// TwinCAT 3 PLC project x_template_xPlc
// Title: x_template_xPlc
// Company: TcOpen.MTS
// ProjectVersion: 0.6.0.913
// ProgramVersion: 3.1.4023.0
// libraries:
//   Tc2_Standard, * (Beckhoff Automation GmbH)
//   Tc2_System, * (Beckhoff Automation GmbH)
//   Tc2_Utilities, * (Beckhoff Automation GmbH)
//   Tc3_Module, * (Beckhoff Automation GmbH)
//   TcoAbbRobotics, 0.12.0.111 (Vortex.Library)
//   TcoAbstractions, 0.12.0.111 (Vortex.Library)
//   TcoAimTtiPowerSupply, 0.12.0.111 (Vortex.Library)
//   TcoCognexVision, 0.12.0.111 (Vortex.Library)
//   TcoCore, 0.12.0.111 (Vortex.Library)
//   TcoData, 0.12.0.111 (Vortex.Library)
//   TcoDrivesBeckhoff, 0.12.0.111 (Vortex.Library)
//   TcoElements, 0.12.0.111 (Vortex.Library)
//   TcoInspectors, 0.12.0.111 (Vortex.Library)
//   TcoIo, 0.12.0.111 (Vortex.Library)
//   TcoKukaRobotics, 0.12.0.111 (Vortex.Library)
//   TcoMitsubishiRobotics, 0.12.0.111 (Vortex.Library)
//   TcoPneumatics, 0.12.0.111 (Vortex.Library)
//   TcoRexrothPress, 0.12.0.111 (Vortex.Library)
//   TcoTixonFeeding, 0.12.0.111 (Vortex.Library)
//   TcoUrRobotics, 0.12.0.111 (Vortex.Library)
//   TcoUtilities, 0.12.0.111 (Vortex.Library)
// project tree:
//   Abstractions/Components/ArrayRenderingExample/ SampleArrayToRender.TcDUT (not stored), SampleDataItem.TcDUT (not stored)
//   Abstractions/Components/MtsFeeding/Blisters/Plb/ TcoPlbPaletizator.TcPOU (not stored), TcoPlbPaletizator_Components.TcDUT (not stored), TcoPlbPaletizator_Config_v_1_x_x.TcDUT (not stored), TcoPlbPaletizator_Control_v_1_x_x.TcDUT (not stored), TcoPlbPaletizator_Positions.TcPOU (not stored), TcoPlbPaletizator_Status_v_1_x_x.TcDUT (not stored)
//   Abstractions/Components/MtsFeeding/Blisters/Plr/ TcoPlrPaletizator.TcPOU (not stored), TcoPlrPaletizator_Components.TcDUT (not stored), TcoPlrPaletizator_Config_v_1_x_x.TcDUT (not stored), TcoPlrPaletizator_Control_v_1_x_x.TcDUT (not stored), TcoPlrPaletizator_Status_v_1_x_x.TcDUT (not stored)
//   Abstractions/Components/MtsFeeding/Blisters/Pls/ TcoPlsPaletizator.TcPOU, TcoPlsPaletizator_Components.TcDUT, TcoPlsPaletizator_Config_v_1_x_x.TcDUT, TcoPlsPaletizator_Control_v_1_x_x.TcDUT (not stored), TcoPlsPaletizator_Status_v_1_x_x.TcDUT
//   Abstractions/Components/MtsFeeding/Blisters/ TcoFeeding_Config_v_1_x_x.TcDUT, TcoFeeding_Status_v_1_x_x.TcDUT
//   Abstractions/Components/MtsFeeding/OscilatingFeeder/ eTcoOscilatingConveyorOscilationModes.TcDUT (not stored), eTcoOscilatingConveyorStatus.TcDUT (not stored), TcoOscilatingConveyorFeeder.TcPOU (not stored), TcoOscilatingConveyorFeederComponents.TcDUT (not stored), TcoOscilatingConveyorFeeder_Config_v_1_x_x.TcDUT (not stored), TcoOscilatingConveyorFeeder_Control_v_1_x_x.TcDUT (not stored), TcoOscilatingConveyorFeeder_DesignerSpecificData.TcPOU (not stored), TcoOscilatingConveyorFeeder_PcToPlc.TcDUT (not stored), TcoOscilatingConveyorFeeder_PlcToPc.TcDUT (not stored), TcoOscilatingConveyorFeeder_Status_v_1_x_x.TcDUT (not stored)
//   Abstractions/Components/MtsFeeding/ TcoFeedingSequenceTask.TcPOU (not stored)
//   Abstractions/Components/Rework/ eReworkResults.TcDUT (not stored), ReworkData.TcDUT (not stored), ReworkInstructionTask.TcPOU (not stored)
//   Abstractions/Components/TS/EqTransfer/ eTcoEq2TransferConfiguration.TcDUT (not stored), eTcoEq2TransferHandlingMode.TcDUT (not stored), TcoEq2Transfer.TcPOU (not stored), TcoEq2TransferComponents.TcDUT (not stored), TcoEq2Transfer_Config.TcDUT (not stored), TcoEq2Transfer_Control.TcDUT (not stored), TcoEq2Transfer_Status.TcDUT (not stored)
//   Abstractions/Components/TS/RotaryTrabsferWithLift/ TcoLiftingRotaryTransfer.TcPOU (not stored), TcoLiftingRotaryTransferComponents.TcDUT (not stored), TcoLiftingRotaryTransfer_Config.TcDUT (not stored), TcoLiftingRotaryTransfer_Control.TcDUT (not stored), TcoLiftingRotaryTransfer_Status.TcDUT (not stored)
//   Abstractions/Components/TS/RotaryTransfer/ TcoRotaryTransfer.TcPOU (not stored), TcoRotaryTransferComponents.TcDUT (not stored), TcoRotaryTransfer_Config.TcDUT (not stored), TcoRotaryTransfer_Control.TcDUT (not stored), TcoRotaryTransfer_Status.TcDUT (not stored)
//   Abstractions/Components/TS/WorkPosition/ TcoTransferSystemComponent.TcPOU (not stored), TcoTransferSystemComponents.TcDUT (not stored), TcoTransferSystem_Config.TcDUT (not stored), TcoTransferSystem_Control.TcDUT (not stored), TcoTransferSystem_Status.TcDUT (not stored)
//   Abstractions/Components/WrappedComponent/ WrappedComponentExample.TcPOU (not stored), WrappedComponentExample_Config.TcDUT (not stored), WrappedComponentExample_Control.TcDUT (not stored), WrappedComponentExample_Status.TcDUT (not stored), WrappedComponentsExample.TcDUT (not stored)
//   Abstractions/CUBase/ CuBaseRecurringFail.TcDUT (not stored), CuBaseRecurringFailures.TcDUT (not stored), CUBase.TcPOU, CUBaseStatusInfo.TcDUT (not stored), CUBaseSettings.TcDUT (not stored), CUComponentsBase.TcDUT, ICUBase.TcIO (not stored), ICUTask.TcIO (not stored), OperatorInfo.TcDUT
//   Abstractions/CUBase/Data/ BasicCounterData.TcDUT (not stored), CuHeader.TcDUT (not stored), CUProcessDataBase.TcDUT (not stored), CUTechnologicalDataBase.TcDUT (not stored), eCUMode.TcDUT (not stored), eCUState.TcDUT (not stored), eDataEntityInvokeType.TcDUT (not stored), EntityHeader.TcDUT (not stored)
//   Abstractions/CUBase/RemoteTasks/ ProductionPlaner.TcPOU (not stored)
//   Abstractions/CUBase/Tasks/ CUBaseAutomat.TcPOU, CUBaseSuspend.TcPOU (not stored), CUBaseGround.TcPOU (not stored), CUBaseRecover.TcPOU (not stored)
//   Abstractions/Generic/LightTower/ TcoLightTower.TcPOU, TcoLightTower_Config.TcDUT (not stored), TcoLightTower_Info.TcDUT (not stored), TcoLightTower_Status.TcDUT (not stored)
//   Abstractions/Generic/NotificationPanel/ eIconType.TcDUT, Icon.TcDUT, NotificationPanel.TcPOU
//   Abstractions/Generic/TagsPairing/ eTagPairingAnswer.TcDUT (not stored), eTagPairingMode.TcDUT (not stored), eTagPairingStatus.TcDUT (not stored), PairTagTask.TcPOU (not stored), TagsPairing.TcDUT (not stored)
//   Abstractions/Safety/ControlButtons/ ITcoControlButtons.TcIO (not stored), TcoControlButtons.TcPOU (not stored), TcoControledZone_Info.TcDUT (not stored), VirtualButtons.TcDUT
//   Abstractions/Safety/ControlledZone/ TcoControlledZone.TcPOU, TcoControlledZoneActionTask.TcPOU (not stored), TcoControlledZone_Config.TcDUT (not stored), TcoControlledZone_Status.TcDUT (not stored)
//   Abstractions/Safety/ControlVoltage/ ITcoControlVoltage.TcIO (not stored), TcoControlVoltage.TcPOU (not stored)
//   Abstractions/Safety/DoorCircuit/ TcoDoorCircuit_Status.TcDUT (not stored), TcoDoorCircuit_Config.TcDUT (not stored), TcoDoorCircuit.TcPOU, ITcoDoorCircuit.TcIO (not stored)
//   Abstractions/Safety/Doors/ ITcoDoorLock.TcIO (not stored), TcoStandardDoor.TcPOU (not stored), TcoBasicDoor.TcPOU (not stored)
//   Abstractions/Safety/Estop/ TcoEmergencyStop.TcPOU (not stored)
//   Abstractions/Safety/KeyMode/ TcoKeyMode_Config.TcDUT (not stored), TcoKeyMode_Status.TcDUT (not stored), TcoKeyMode.TcPOU (not stored), ITcoKeyMode.TcIO (not stored)
//   Abstractions/Safety/KeyNormalService/ TcoKeyNormalService.TcPOU (not stored), ITcoKeyNormalSevice.TcIO (not stored)
//   Abstractions/TcoCore/ CycleTimeAnalitics.TcDUT (not stored), TcoCustomExportSeqData.TcDUT, TcoCustomStepDetails.TcDUT, TcoCustomTimeStruct.TcDUT, TcoInnerTask.TcPOU (not stored), TcoCustomSequencerObserver.TcPOU, TcoTaskedSequencer.TcPOU, TcoTaskedService.TcPOU (not stored)
//   Abstractions/Technology/ eStations.TcDUT
//   / MAIN.TcPOU (not stored), PlcTask.TcTTO (not stored)
//   Technology/CU00x/Automat/ CU00xAutomatParalell_1_Task.TcPOU, CU00xAutomatTask.TcPOU
//   Technology/CU00x/Components/ CU00xExamplesOfComponents.TcDUT (not stored), CU00xComponents.TcDUT
//   Technology/CU00x/Data/ CU00xTechnologicalData.TcDUT (not stored), CU00xDialogContent.TcPOU (not stored), CU00xProcessData.TcDUT
//   Technology/CU00x/Ground/ CU00xGroundTask.TcPOU (not stored)
//   Technology/CU00x/Manual/ CU00xManualTask.TcPOU (not stored)
//   Technology/CU00x/Positions/ CU00xTestMultiPositions.TcPOU (not stored), Cu00xTestPositions.TcPOU (not stored)
//   Technology/CU00x/Safety/Suspend/ CU00xSuspendTask.TcPOU
//   Technology/CU00x/Safety/Recover/ CU00xRecoverTask.TcPOU
//   Technology/Data/ InternalStorage.TcPOU, ProcessData.TcDUT, ProcessDataManager.TcPOU (not stored), TcoEntityBase.TcDUT (not stored), TechnologicalDataManager.TcPOU (not stored), TechnologyData.TcDUT
//   Technology/CU00x/ CU00x.TcPOU (not stored)
//   Technology/ Technology.TcPOU, TechnologyComponents.TcDUT
//   DUTs/IO/PDOs/ Device_State_F0482DC3.TcDUT (not stored), Device_Control_6258066A.TcDUT (not stored), Inputs_23559BB0.TcDUT (not stored), Outputs_FC2FACAD.TcDUT (not stored), Modules_85784B27.TcDUT (not stored), Channel_830843C1.TcDUT (not stored), Channel_42CA91F7.TcDUT (not stored)
//   DUTs/IO/Boxes/ EK1200_013D0B49.TcDUT (not stored), EK1122_1FC0878B.TcDUT (not stored), AES_510494FB.TcDUT (not stored), EPP1322_1FC0878B.TcDUT (not stored), EPP1809_32157CFD.TcDUT (not stored), EPP1008_78E8D3DD.TcDUT (not stored), EL1809_32157CFD.TcDUT (not stored), EL2809_2B6483BD.TcDUT (not stored), EL9011_D65D3D32.TcDUT (not stored)
//   DUTs/IO/Devices/ SyncUnitTasks_4BE01469.TcDUT (not stored), SyncUnits_67D36DDA.TcDUT (not stored)
//   DUTs/IO/Topology/ EK_E812B8FA.TcDUT (not stored), EC_4E5C738F.TcDUT (not stored), EC_245FBB9A.TcDUT (not stored)
//   GVLs/ GVL_iXlinker.TcGVL (not stored)
// real-time tasks:
//   TASK PlcTask: cycle T#10ms, priority 20, ADS port 350
//   TASK PlcTask1: cycle T#10ms, priority 21, ADS port 351
// I/O:
//   DEVICE EC1 (disabled), AmsNetId 192.168.4.1.7.1
//     (EK1200) [EK1200-5000 EtherCAT Power supply (2A E-Bus)]
//       EC (EK1122) [EK1122 2 port EtherCAT junction]
//       PN (EL6631) [EL6631 PROFINET IO Controller]
//       IA1 (EL1809) [EL1809 16Ch. Dig. Input 24V, 3ms]
//       QA1 (EL2809) [EL2809 16Ch. Dig. Output 24V, 0.5A]
//       Term 6 (EL4004) [EL4004 4Ch. Ana. Output 0-10V, 12bit]
//       Term 7 (EL7342) [EL7342 2Ch. DC motor output stage (50V, 3.5A)]
//       Term 8 (EL4004) [EL4004 4Ch. Ana. Output 0-10V, 12bit]
//       Term 9 (EL6001) [EL6001 Interface (RS232)]
//       Term 13 (EL9011) [EL9011 End Terminal]
//   DEVICE EC (disabled), AmsNetId 192.168.4.1.2.1
//     EC [EK1200-5000 EtherCAT Power supply (2A E-Bus)]
//       EK [EK1122 2 port EtherCAT junction]
//         PNEU [AES Fieldbus Coupler Gen2]
//           modules: Modules
//         AB [EPP1322-0001 3 port EtherCAT P gateway]
//         AB21 [EPP1809-0021 16 Ch. Dig. Input 24V, 3ms, M8]
//         AB22 [EPP1809-0021 16 Ch. Dig. Input 24V, 3ms, M8]
//         AB23 [EPP1008-0001 8 Ch. Dig. Input 24V, 3ms, M8]
//         AB24 [EPP1008-0001 8 Ch. Dig. Input 24V, 3ms, M8]
//       IA1 [EL1809 16Ch. Dig. Input 24V, 3ms]
//       QA1 [EL2809-0015 16Ch. Dig. Output 24V DC, 0.35A, not short-circuit proof]
//       Term 11 (EL9011) [EL9011 End Terminal]
// variable links:
//   x_template_xPlc/x_template_xPlc Instance <-> EC
//     PlcTask Inputs/GVL_iXlinker.EC.InfoData.AmsNetId <-> InfoData/AmsNetId
//     PlcTask Inputs/GVL_iXlinker.EC.InfoData.CfgSlaveCount <-> InfoData/CfgSlaveCount
//     PlcTask Inputs/GVL_iXlinker.EC.InfoData.ChangeCount <-> InfoData/ChangeCount
//     PlcTask Inputs/GVL_iXlinker.EC.InfoData.DevId <-> InfoData/DevId
//     PlcTask Inputs/GVL_iXlinker.EC.Inputs.DevState <-> Inputs/DevState
//     PlcTask Inputs/GVL_iXlinker.EC.Inputs.Frm0InputToggle <-> Inputs/Frm0InputToggle
//     PlcTask Inputs/GVL_iXlinker.EC.Inputs.Frm0State <-> Inputs/Frm0State
//     PlcTask Inputs/GVL_iXlinker.EC.Inputs.Frm0WcState <-> Inputs/Frm0WcState
//     PlcTask Inputs/GVL_iXlinker.EC.Inputs.SlaveCount <-> Inputs/SlaveCount
//     PlcTask Outputs/GVL_iXlinker.EC.Outputs.DevCtrl <-> Outputs/DevCtrl
//     PlcTask Outputs/GVL_iXlinker.EC.Outputs.Frm0Ctrl <-> Outputs/Frm0Ctrl
//     PlcTask Outputs/GVL_iXlinker.EC.Outputs.Frm0WcCtrl <-> Outputs/Frm0WcCtrl
//   x_template_xPlc/x_template_xPlc Instance <-> EC/EC/EK
//     PlcTask Inputs/GVL_iXlinker.EC.EC.EK.InfoData.State <-> InfoData/State
//   x_template_xPlc/x_template_xPlc Instance <-> EC/EC/EK/AB
//     PlcTask Inputs/GVL_iXlinker.EC.EC.EK.AB.InfoData.State <-> InfoData/State
//   x_template_xPlc/x_template_xPlc Instance <-> EC/EC/EK/AB21
//     PlcTask Inputs/GVL_iXlinker.EC.EC.EK.AB21.Channel_{1..16}.Input <-> Channel {1..16}/Input  (16 links)
//     PlcTask Inputs/GVL_iXlinker.EC.EC.EK.AB21.InfoData.State <-> InfoData/State
//     PlcTask Inputs/GVL_iXlinker.EC.EC.EK.AB21.WcState.InputToggle <-> WcState/InputToggle
//     PlcTask Inputs/GVL_iXlinker.EC.EC.EK.AB21.WcState.WcState <-> WcState/WcState
//   x_template_xPlc/x_template_xPlc Instance <-> EC/EC/EK/AB22
//     PlcTask Inputs/GVL_iXlinker.EC.EC.EK.AB22.Channel_{1..16}.Input <-> Channel {1..16}/Input  (16 links)
//     PlcTask Inputs/GVL_iXlinker.EC.EC.EK.AB22.InfoData.State <-> InfoData/State
//     PlcTask Inputs/GVL_iXlinker.EC.EC.EK.AB22.WcState.InputToggle <-> WcState/InputToggle
//     PlcTask Inputs/GVL_iXlinker.EC.EC.EK.AB22.WcState.WcState <-> WcState/WcState
//   x_template_xPlc/x_template_xPlc Instance <-> EC/EC/EK/AB23
//     PlcTask Inputs/GVL_iXlinker.EC.EC.EK.AB23.Channel_{1..8}.Input <-> Channel {1..8}/Input  (8 links)
//     PlcTask Inputs/GVL_iXlinker.EC.EC.EK.AB23.InfoData.State <-> InfoData/State
//     PlcTask Inputs/GVL_iXlinker.EC.EC.EK.AB23.WcState.InputToggle <-> WcState/InputToggle
//     PlcTask Inputs/GVL_iXlinker.EC.EC.EK.AB23.WcState.WcState <-> WcState/WcState
//   x_template_xPlc/x_template_xPlc Instance <-> EC/EC/EK/AB24
//     PlcTask Inputs/GVL_iXlinker.EC.EC.EK.AB24.Channel_{1..8}.Input <-> Channel {1..8}/Input  (8 links)
//     PlcTask Inputs/GVL_iXlinker.EC.EC.EK.AB24.InfoData.State <-> InfoData/State
//     PlcTask Inputs/GVL_iXlinker.EC.EC.EK.AB24.WcState.InputToggle <-> WcState/InputToggle
//     PlcTask Inputs/GVL_iXlinker.EC.EC.EK.AB24.WcState.WcState <-> WcState/WcState
//   x_template_xPlc/x_template_xPlc Instance <-> EC/EC/EK/PNEU
//     PlcTask Inputs/GVL_iXlinker.EC.EC.EK.PNEU.Device_State.CommonValve <-> Device_State/CommonValve
//     PlcTask Inputs/GVL_iXlinker.EC.EC.EK.PNEU.Device_State.Configuration_Error_IO_Module <-> Device_State/Configuration Error IO-Module
//     PlcTask Inputs/GVL_iXlinker.EC.EC.EK.PNEU.Device_State.Configuration_Error_Valve <-> Device_State/Configuration Error Valve
//     PlcTask Inputs/GVL_iXlinker.EC.EC.EK.PNEU.Device_State.Configuratipn_Error_SLS <-> Device_State/Configuratipn Error SLS
//     PlcTask Inputs/GVL_iXlinker.EC.EC.EK.PNEU.Device_State.Count_IO_Module_to_big <-> Device_State/Count IO-Module to big
//     PlcTask Inputs/GVL_iXlinker.EC.EC.EK.PNEU.Device_State.Heardbeat_x <-> Device_State/Heardbeat
//     PlcTask Inputs/GVL_iXlinker.EC.EC.EK.PNEU.Device_State.IO_1_8 <-> Device_State/IO:1-8
//     PlcTask Inputs/GVL_iXlinker.EC.EC.EK.PNEU.Device_State.IO_9_10 <-> Device_State/IO:9-10
//     PlcTask Inputs/GVL_iXlinker.EC.EC.EK.PNEU.Device_State.Switchcounter_Error <-> Device_State/Switchcounter Error
//     PlcTask Inputs/GVL_iXlinker.EC.EC.EK.PNEU.Device_State.UA_OFF <-> Device_State/UA OFF
//     PlcTask Inputs/GVL_iXlinker.EC.EC.EK.PNEU.Device_State.UL_OFF <-> Device_State/UL OFF
//     PlcTask Inputs/GVL_iXlinker.EC.EC.EK.PNEU.Device_State.Undervoltage_5V <-> Device_State/Undervoltage 5V
//     PlcTask Inputs/GVL_iXlinker.EC.EC.EK.PNEU.Device_State.Undervoltage_UA <-> Device_State/Undervoltage UA
//     PlcTask Inputs/GVL_iXlinker.EC.EC.EK.PNEU.Device_State.Undervoltage_UL <-> Device_State/Undervoltage UL
//     PlcTask Inputs/GVL_iXlinker.EC.EC.EK.PNEU.Device_State.Unknown_Module_ID <-> Device_State/Unknown Module ID
//     PlcTask Inputs/GVL_iXlinker.EC.EC.EK.PNEU.Device_State.ValveExtSupplyDiag_1_6 <-> Device_State/ValveExtSupplyDiag:1-6
//     PlcTask Inputs/GVL_iXlinker.EC.EC.EK.PNEU.InfoData.AdsAddr <-> InfoData/AdsAddr
//     PlcTask Inputs/GVL_iXlinker.EC.EC.EK.PNEU.InfoData.State <-> InfoData/State
//     PlcTask Inputs/GVL_iXlinker.EC.EC.EK.PNEU.Modules.Inputs.digital_Data_I[{0..31}] <-> Modules/Inputs/digital Data I_{0..31}  (32 links)
//     PlcTask Inputs/GVL_iXlinker.EC.EC.EK.PNEU.WcState.InputToggle <-> WcState/InputToggle
//     PlcTask Inputs/GVL_iXlinker.EC.EC.EK.PNEU.WcState.WcState <-> WcState/WcState
//     PlcTask Outputs/GVL_iXlinker.EC.EC.EK.PNEU.Device_Control.Default_Modul_Control <-> Device_Control/Default_Modul_Control
//     PlcTask Outputs/GVL_iXlinker.EC.EC.EK.PNEU.Device_Control.Freeze_Output <-> Device_Control/Freeze Output
//     PlcTask Outputs/GVL_iXlinker.EC.EC.EK.PNEU.Device_Control.HL_Swap <-> Device_Control/HL_Swap
//     PlcTask Outputs/GVL_iXlinker.EC.EC.EK.PNEU.Device_Control.Web_App_Disable <-> Device_Control/Web App Disable
//     PlcTask Outputs/GVL_iXlinker.EC.EC.EK.PNEU.Modules.Outputs.digital_Data_O[{0..31}] <-> Modules/Outputs/digital Data O_{0..31}  (32 links)
//   x_template_xPlc/x_template_xPlc Instance <-> EC/EC/IA1
//     PlcTask Inputs/GVL_iXlinker.EC.EC.IA1.Channel_{1..16}.Input <-> Channel {1..16}/Input  (16 links)
//     PlcTask Inputs/GVL_iXlinker.EC.EC.IA1.InfoData.State <-> InfoData/State
//     PlcTask Inputs/GVL_iXlinker.EC.EC.IA1.WcState.InputToggle <-> WcState/InputToggle
//     PlcTask Inputs/GVL_iXlinker.EC.EC.IA1.WcState.WcState <-> WcState/WcState
//   x_template_xPlc/x_template_xPlc Instance <-> EC/EC/QA1
//     PlcTask Inputs/GVL_iXlinker.EC.EC.QA1.InfoData.State <-> InfoData/State
//     PlcTask Inputs/GVL_iXlinker.EC.EC.QA1.WcState.WcState <-> WcState/WcState
//     PlcTask Outputs/GVL_iXlinker.EC.EC.QA1.Channel_{1..16}.Output <-> Channel {1..16}/Output  (16 links)

// ---- Abstractions/Components/MtsFeeding/Blisters/Pls/TcoPlsPaletizator_Components.TcDUT
TYPE TcoPlsPaletizator_Components EXTENDS TcoCore.TcoStruct:
STRUCT
	
	{attribute wpf [Container(Layout.Stack)]}
	{attribute addProperty Name "(I1) <#Blister present in entry slide#>"}
	I1_PresentBlisterEntry : TcoElements.TcoDi(THISSTRUCT);
	
	{attribute addProperty Name "(I2) <#Gap detected between blisters#>"}
	I2_PresentBlisterEntryEmptySpace : TcoElements.TcoDi(THISSTRUCT);
	
	{attribute addProperty Name "(I3) <#Blister feeder empty#>"}
	I3_PresentBlistersInBufferEmpty : TcoElements.TcoDi(THISSTRUCT);

	
	{attribute addProperty Name "(I4) <#Blister in working position#>"}
	I4_PresentBlisterInWorkingPos : TcoElements.TcoDi(THISSTRUCT);
		
	{attribute addProperty Name "(I5) <#Output blister not on slide conveyor#>"}
	I5_OutBlistersIsThrowedCorrectly : TcoElements.TcoDi(THISSTRUCT);
	
	{attribute addProperty Name "(I6) <#Output blister present in elevator#>"}
	I6_OutBlistersLisftSignal : TcoElements.TcoDi(THISSTRUCT);
	
	{attribute addProperty Name "(I7) <#Output blister above buffer#>"}
	I7_OutBlistersIsAboveOutBuffer : TcoElements.TcoDi(THISSTRUCT);
	
	{attribute addProperty Name "(I8) <#Output container full#>"}
	I8_OutBlistersBufferIsFull : TcoElements.TcoDi(THISSTRUCT);
	
	
	{attribute wpf [Container(Layout.Stack)]}
	{attribute addProperty Name "(P1) <#Entry blister lift#>"}
	P1_VerticalSepareEntryBlisters : TcoPneumatics.TcoCylinder(THISSTRUCT);
	
	{attribute addProperty Name "(P2) <#Entry blister lift#>"}
	P2_VerticalSepareEntryBlisters : TcoPneumatics.TcoCylinder(THISSTRUCT);
	
	{attribute addProperty Name "(P3) (P3.1) <#Entry blister slide#>"}
	P3_HorizontalSepareEntryBlisters : TcoPneumatics.TcoDoubleCylinder(THISSTRUCT);
		
	{attribute addProperty Name "(P4) <#Entry blister feed#>"}
	P4_FeedEntryBlister :TcoPneumatics.TcoCylinder(THISSTRUCT);
	
	{attribute addProperty Name "(P5) (P5.1) <#Output blister slide#>"}
	P5_HorizontalSepareOutBlisters : TcoPneumatics.TcoDoubleCylinder(THISSTRUCT);
	
	{attribute addProperty Name "(P6) <#Output blister lift#>"}
	P6_VerticalSepareOutBlister : TcoPneumatics.TcoCylinder(THISSTRUCT);
	
	{attribute addProperty Name "(P7) <#Entry blister support#>"}
	P7_SupportEntryBlister : TcoPneumatics.TcoCylinder(THISSTRUCT);
	
	{attribute addProperty Name "(P8) (P8.1) <#Entry blister side clamp#>"}
	P8_FixEntryBlisterSide : TcoPneumatics.TcoDoubleCylinder(THISSTRUCT);
	
	{attribute addProperty Name "(P9) (P9.1) <#Entry blister top clamp#>"}
	P9_LockEntryBlisterTop : TcoPneumatics.TcoDoubleCylinder(THISSTRUCT);
	
	{attribute addProperty Name "(P10) (P10.1) <#Entry blister separator#>"}
	P10_HoldEntrySepareOutBlister : TcoPneumatics.TcoDoubleCylinder(THISSTRUCT);
	
	
	
	{attribute wpf [Container(Layout.Stack,"Vseobecne")]}
	
	{attribute addProperty Name "(Q1) <#Warning signalisation#> R"}
	Q1_AttentionSignalisationR : TcoElements.TcoDo(THISSTRUCT);
	{attribute addProperty Name "(Q2) <#Warning signalisation#> G"}
	Q2_AttentionSignalisationG : TcoElements.TcoDo(THISSTRUCT);
	{attribute addProperty Name "(Q3) <#Warning signalisation#> B"}
	Q3_AttentionSignalisationB : TcoElements.TcoDo(THISSTRUCT);

	
	
END_STRUCT
END_TYPE

// ---- Abstractions/Components/MtsFeeding/Blisters/Pls/TcoPlsPaletizator_Config_v_1_x_x.TcDUT
TYPE
    TcoPlsPaletizator_Config_v_1_x_x EXTENDS TcoFeeding_Config_v_1_x_x :
    STRUCT

		
		
        {attribute addProperty Name "<#Locking of the blister from above inactive (P9)(P9.1) is not present#>"}
		LockBlisterInPickPosInactive : BOOL;
		
		{attribute addProperty Name "<#Separation of entry blisters inactive (P10)(P10.1) is not present#>"}
		SepareBlistersAtEntryInactive : BOOL;

    END_STRUCT
END_TYPE

// ---- Abstractions/Components/MtsFeeding/Blisters/Pls/TcoPlsPaletizator_Status_v_1_x_x.TcDUT
TYPE
    TcoPlsPaletizator_Status_v_1_x_x EXTENDS TcoFeeding_Status_v_1_x_x:
    STRUCT

        {attribute addProperty Name "<#Refill required#>"}
		EntryBufferEmpty:BOOL;
		
		{attribute addProperty Name "<#Blister ready#>"}
        BlisterReady : BOOL;
		
		{attribute addProperty Name "<#Empty blisters removal required#>"}
        OutBufferFull : BOOL;
    END_STRUCT
END_TYPE

// ---- Abstractions/Components/MtsFeeding/Blisters/TcoFeeding_Config_v_1_x_x.TcDUT
TYPE
    TcoFeeding_Config_v_1_x_x EXTENDS TcoCore.TcoStruct :
    STRUCT

		{attribute addProperty Name "<#Info delay#>"}
        InfoTime : TIME := T#5S;
		{attribute addProperty Name "<#Error delay#>"}
        ErrorTime : TIME := T#0S;
        {attribute addProperty Name "<#Stabilisation time#>"}
        StabilisationTime : TIME := T#500MS;
        {attribute addProperty Name "<#Blink period#> "}
        BlinkTime : TIME := T#500MS;

        {attribute addProperty Name "<#Safety disable duration#> "}
        TimeToDisableSafety : TIME := T#10S;

        {attribute addProperty Name "<#Step mode managable from outside#> (SetSequencesToStep)"}
        StepModeManagableFromOutside : BOOL;

    END_STRUCT
END_TYPE

// ---- Abstractions/Components/MtsFeeding/Blisters/TcoFeeding_Status_v_1_x_x.TcDUT
TYPE
    TcoFeeding_Status_v_1_x_x EXTENDS TcoCore.TcoStruct :
    STRUCT

	
		{attribute addProperty Name "<#Action#>"}
        ActionDescription : STRING;
		
		{attribute addProperty Name "<#Safety conditon met#>"}
        SafeCondition : BOOL;

    END_STRUCT
END_TYPE

// ---- Abstractions/CUBase/CUComponentsBase.TcDUT
TYPE
    CUComponentsBase EXTENDS TcoCore.TcoStruct :
    STRUCT
       	{attribute wpf [Container(Layout.Stack)]}
		{attribute clr [RenderIgnore()]}
        DummyCylinder : TcoPneumatics.TcoCylinder(THISSTRUCT);
		{attribute clr [RenderIgnore()]}
        DummyDi : TcoElements.TcoDi(THISSTRUCT);
		{attribute clr [RenderIgnore()]}
        DummyDo : TcoElements.TcoDo(THISSTRUCT);
    END_STRUCT
END_TYPE

// ---- Abstractions/CUBase/OperatorInfo.TcDUT
TYPE OperatorInfo EXTENDS TcoCore.TcoStruct :
STRUCT
	UserName : STRING(255);
	
END_STRUCT
END_TYPE

// ---- Abstractions/Generic/NotificationPanel/eIconType.TcDUT
{attribute 'qualified_only'}
{attribute 'strict'}
{attribute 'to_string'}
TYPE 
	eIconType : 
(
	None                 := 0,
	ControlVoltage       := 10,
	AirPressure          := 20,
	EmergencyStop        := 30,
	SafetyDoor           := 40,
	DoorClosed           := 50,
	DoorLocked           := 60,
	AutomatAllowed       := 70,
	ProcessDataLoaded    := 80,
	TechnologyDataLoaded := 90,
	OpticBarrier         := 100,
	Robot                := 110,
	PlcConnection        := 120
);
END_TYPE

// ---- Abstractions/Generic/NotificationPanel/Icon.TcDUT
TYPE Icon :
STRUCT
	Title : STRING;
	IconType : STRING;
	Signal : BOOL;
	BlinkingEnabled : BOOL := FALSE;
	EnableRedIcon : BOOL := TRUE;
	
	///used internally
	SignalBlink : BOOL;
END_STRUCT
END_TYPE

// ---- Abstractions/Safety/ControlButtons/VirtualButtons.TcDUT
TYPE VirtualButtons :
STRUCT
	StartButton:BOOL;
	StopButton:BOOL;
	GroundButton:BOOL;
	AutomatButton:BOOL;

	StartLight : BOOL;
	StopLight : BOOL;
END_STRUCT
END_TYPE

// ---- Abstractions/TcoCore/TcoCustomExportSeqData.TcDUT
TYPE
    TcoCustomExportSeqData :
    STRUCT

        Steps : ARRAY[0..TcoCustomSequencerObserver.MAX_STEPS] OF TcoCustomStepDetails;
        CycleId : STRING(254);
        CuId : UINT;
        StartTime : TcoCustomTimeStruct;
        EndTime : TcoCustomTimeStruct;
    END_STRUCT
END_TYPE

// ---- Abstractions/TcoCore/TcoCustomStepDetails.TcDUT

TYPE TcoCustomStepDetails :
STRUCT

	{attribute addProperty Name "<#Step ID#>"}
	ID: INT;

	{attribute addProperty Name "<#Step description#>"}
	Description: STRING(254);

	{attribute addProperty Name "<#Step duration#>"}
	Duration : TIME;
	
	{attribute addProperty Name "<#Time Stamp Struct#>"}
	TimeStamp : TcoCustomTimeStruct;
	
END_STRUCT
END_TYPE

// ---- Abstractions/TcoCore/TcoCustomTimeStruct.TcDUT
TYPE
    TcoCustomTimeStruct :
    STRUCT
        Year : WORD;
        Month : WORD;

        Day : WORD;
        Hour : WORD;
        Minute : WORD;
        Second : WORD;
        Milliseconds : WORD;
    END_STRUCT
END_TYPE

// ---- Abstractions/Technology/eStations.TcDUT
{attribute 'qualified_only'}
{attribute 'strict'}
TYPE
    eStations :
    (
		CU00x := 100,
       CU010  := 1,
        CU020  := 2,
        CU030  := 3,
        CU040  := 4,
        CU050  := 5,
        ST_6  := 6,
        ST_7  := 7,
        ST_8  := 8,
        ST_9  := 9,
        ST_10 := 10,
        ST_11 := 11,
        ST_12 := 12,
        ST_13 := 13,
        ST_14 := 14,
        ST_15 := 15,
        ST_16 := 16,
        ST_17 := 17,
        ST_18 := 18,
        ST_19 := 19,
        ST_20 := 20,
        NONE  := 32767
    );
END_TYPE

// ---- Technology/Data/ProcessData.TcDUT
{attribute clr [Container(Layout.Tabs)]}
TYPE
    ProcessData EXTENDS TcoEntityBase :
    STRUCT

        {attribute addProperty Name "<#Entity header#>"}
        EntityHeader : EntityHeader     := (Parent := THISSTRUCT);
		{attribute addProperty Name "<#CU00x#>"}
		{attribute clr [Container(Layout.Stack)]}
        CU00x : CU00xProcessData := (Parent := THISSTRUCT);
		
//		
		CU010 : CU010ProcessData := (Parent := THISSTRUCT);
		CU020 : CU020ProcessData := (Parent := THISSTRUCT);
		CU030 : CU030ProcessData := (Parent := THISSTRUCT);
		CU040 : CU040ProcessData := (Parent := THISSTRUCT);
		CU050 : CU050ProcessData := (Parent := THISSTRUCT);
    END_STRUCT
END_TYPE

// ---- Technology/CU00x/Components/CU00xComponents.TcDUT
{attribute wpf [Container(Layout.Tabs)]}
TYPE
    CU00xComponents EXTENDS CUComponentsBase :
    STRUCT
		{attribute wpf [Container(Layout.Stack)]}
		{attribute wpf [Group(Layout.Scroll)]}
		{attribute addProperty Name "Supplu TTI QL"}
     	Supply : TcoAimTtiPowerSupply.TcoQl355P_v_1_x_x (THISSTRUCT);
		{attribute wpf [Container(Layout.Stack)]}
		PairTagTask: PairTagTask(THISSTRUCT);
		{attribute wpf [Container(Layout.Stack)]}
		{attribute addProperty Name "<#ReworkInstruction#>"}
		ReworkInstructionTask : ReworkInstructionTask(THISSTRUCT);
		{attribute wpf [Container(Layout.Stack,"DRIVES AND MANIPULATORS")]}	
		{attribute wpf [Group(Layout.Scroll)]}
		{attribute addProperty Name "MultiAxis"}
     	MultiAxis : TcoDrivesBeckhoff.TcoMultiAxis(THISSTRUCT);
		{attribute addProperty Name "Single Axis"}
     	SingleAxis : TcoDrivesBeckhoff.TcoSingleAxis(THISSTRUCT);
		{attribute addProperty Name "Simple drive"}
     	SimpleDrive : TcoDrivesBeckhoff.TcoDriveSimple(THISSTRUCT);
		
		{attribute wpf [Container(Layout.Stack,"VISION")]}	
		{attribute wpf [Group(Layout.Scroll)]}
		{attribute addProperty Name "Dataman"}
     	Dmc : TcoCognexVision.TcoDataman_v_5_x_x(THISSTRUCT);
		{attribute addProperty Name "Insight"}
     	Cam : TcoCognexVision.TcoInsight_v_5_x_x(THISSTRUCT);

	
		{attribute wpf [Container(Layout.Stack,"ROBOTICS")]}	
		{attribute wpf [Group(Layout.Scroll)]}
		{attribute addProperty Name "Abb IRC 5"}
     	AbbIrc5 : TcoAbbRobotics.TcoIrc5_v_1_x_x(THISSTRUCT);
		{attribute addProperty Name "Abb Omnicore"}
     	AbbOmnicore : TcoAbbRobotics.TcoOmnicore_v_1_x_x(THISSTRUCT);
		
		{attribute addProperty Name "Mitshubishi Cr series"}
     	MitshubishiCr: TcoMitsubishiRobotics.TcoCr800_v_1_x_x(THISSTRUCT);
		{attribute addProperty Name "UR CB series"}
     	UrCb3:  TcoUrRobotics.TcoUrCb3_v_3_x_x(THISSTRUCT);
		{attribute addProperty Name "Ur E series"}
     	UrEseries: TcoUrRobotics.TcoUrEseries_v_5_x_x(THISSTRUCT);
		
		{attribute addProperty Name "Kuka Krc4"}
     	KukaKrc4: TcoKukaRobotics.TcoKrc4_v_5_x_x(THISSTRUCT);
		
		{attribute wpf [Container(Layout.Stack,"TIXONS")]}	
		{attribute wpf [Group(Layout.Scroll)]}
		{attribute addProperty Name "Tixon Vibro"}
     	TixonVibro : TcoTixonFeeding.TcoTixonVibro_v_1_x_x(THISSTRUCT);
		{attribute addProperty Name "Tixon Step"}
     	TixonStep : TcoTixonFeeding.TcoTixonStep_v_1_x_x(THISSTRUCT);
		
		{attribute addProperty Name "Tixon Pick Vibro"}
     	TixonPickVibro : TcoTixonFeeding.TcoTixonPickVibro_v_1_x_x(THISSTRUCT);
		{attribute addProperty Name "Tixon Pick Step"}
     	TixonPickStep : TcoTixonFeeding.TcoTixonPickStep_v_1_x_x(THISSTRUCT);
			
		{attribute wpf [Container(Layout.Stack,"MtsFeeding")]}	
		{attribute wpf [Group(Layout.Scroll)]}
		PlsPaletizator:TcoPlsPaletizator(THISSTRUCT);	
		{attribute clr [RenderIgnore()]}
		PlsPaletizatorComponents:TcoPlsPaletizator_Components := (Parent := THISSTRUCT);  
		
		{attribute wpf [Group(Layout.Scroll)]}
		PlrPaletizator:TcoPlrPaletizator(THISSTRUCT);	
		{attribute clr [RenderIgnore()]}
		PlrPaletizatorComponents:TcoPlrPaletizator_Components := (Parent := THISSTRUCT);  
		
		{attribute wpf [Group(Layout.Scroll)]}
		PlbPaletizator:TcoPlbPaletizator(THISSTRUCT);	
		{attribute clr [RenderIgnore()]}
		PlbPaletizatorComponents:TcoPlbPaletizator_Components := (Parent := THISSTRUCT);  
		
		
		{attribute wpf [Container(Layout.Stack)]}
        {attribute wpf [Group(Layout.Scroll)]}
        OscilatingFeeder : TcoOscilatingConveyorFeeder(THISSTRUCT);
        {attribute clr [RenderIgnore()]}
        OscilatingFeederComponents : TcoOscilatingConveyorFeederComponents := (Parent := THISSTRUCT);

		
		{attribute wpf [Container(Layout.Stack,"Wrapped component example")]}	
		{attribute wpf [Group(Layout.Scroll)]}
		PickAndPlace:WrappedComponentExample(THISSTRUCT);
		{attribute wpf [Container(Layout.Stack,"Wrapped component struct")]}	
		PickAndPlaceCompoennts:WrappedComponentsExample := (Parent := THISSTRUCT);  

		{attribute addProperty Name "GROUP 1"}
		Group1 : CU00xExamplesOfComponents := (Parent := THISSTRUCT);  
		{attribute addProperty Name "GROUP 2"}
		Group2 : CU00xExamplesOfComponents := (Parent := THISSTRUCT); 
 
		
		
		{attribute wpf [Container(Layout.Stack,"PanaTrace")]}	
		{attribute wpf [Group(Layout.Scroll)]}
		PanaTrace:TcoPscPanaTrace(THISSTRUCT);
    END_STRUCT
END_TYPE

// ---- Technology/CU00x/Data/CU00xProcessData.TcDUT
TYPE
    CU00xProcessData EXTENDS CUProcessDataBase :
    STRUCT
		{attribute wpf [Container(Layout.Stack)]}
		{attribute addProperty Name "Bolt present inspection"}
        BoltPresenceInspector : TcoInspectors.TcoDigitalInspector(THISSTRUCT);
		{attribute addProperty Name "Bolt Dimension inspection"}
		BoltDimensionPresenceInspector : TcoInspectors.TcoAnalogueInspector(THISSTRUCT);
		{attribute addProperty Name "Bolt code inspection"}
		BoltDatacodePresenceInspector : TcoInspectors.TcoDataInspector(THISSTRUCT);
		

		{attribute addProperty Name "Dimension inspection 1"}
        Dim_Inspector_1 : TcoInspectors.TcoAnalogueInspector(THISSTRUCT);
		{attribute addProperty Name "Dimension inspection 2"}
        Dim_Inspector_2 : TcoInspectors.TcoAnalogueInspector(THISSTRUCT);
		{attribute addProperty Name "Dimension inspection 3"}
		Dim_Inspector_3 : TcoInspectors.TcoAnalogueInspector(THISSTRUCT);
		{attribute addProperty Name "Dimension inspection 4"}
        Dim_Inspector_4 : TcoInspectors.TcoAnalogueInspector(THISSTRUCT);
		{attribute addProperty Name "Dimension inspection 5"}
        Dim_Inspector_5 : TcoInspectors.TcoAnalogueInspector(THISSTRUCT);
		{attribute addProperty Name "Dimension inspection 6"}
        Dim_Inspector_6 : TcoInspectors.TcoAnalogueInspector(THISSTRUCT);
		{attribute addProperty Name "Dimension inspection 7"}
        Dim_Inspector_7 : TcoInspectors.TcoAnalogueInspector(THISSTRUCT);
		{attribute addProperty Name "Dimension inspection 8"}
        Dim_Inspector_8 : TcoInspectors.TcoAnalogueInspector(THISSTRUCT);
		{attribute addProperty Name "Dimension inspection 9"}
        Dim_Inspector_9 : TcoInspectors.TcoAnalogueInspector(THISSTRUCT);
		{attribute addProperty Name "Dimension inspection 10"}
        Dim_Inspector_10 : TcoInspectors.TcoAnalogueInspector(THISSTRUCT);
		
		{attribute addProperty Name "Dimension inspection 11"}
        Dim_Inspector_11 : TcoInspectors.TcoAnalogueInspector(THISSTRUCT);
		{attribute addProperty Name "Dimension inspection 12"}
        Dim_Inspector_12 : TcoInspectors.TcoAnalogueInspector(THISSTRUCT);
		{attribute addProperty Name "Dimension inspection 13"}
		Dim_Inspector_13 : TcoInspectors.TcoAnalogueInspector(THISSTRUCT);
		{attribute addProperty Name "Dimension inspection 14"}
        Dim_Inspector_14 : TcoInspectors.TcoAnalogueInspector(THISSTRUCT);
		{attribute addProperty Name "Dimension inspection 15"}
        Dim_Inspector_15 : TcoInspectors.TcoAnalogueInspector(THISSTRUCT);
		{attribute addProperty Name "Dimension inspection 16"}
        Dim_Inspector_16 : TcoInspectors.TcoAnalogueInspector(THISSTRUCT);
		{attribute addProperty Name "Dimension inspection 17"}
        Dim_Inspector_17 : TcoInspectors.TcoAnalogueInspector(THISSTRUCT);
		{attribute addProperty Name "Dimension inspection 18"}
        Dim_Inspector_18 : TcoInspectors.TcoAnalogueInspector(THISSTRUCT);
		{attribute addProperty Name "Dimension inspection 19"}
        Dim_Inspector_19 : TcoInspectors.TcoAnalogueInspector(THISSTRUCT);
		{attribute addProperty Name "Dimension inspection 20"}
        Dim_Inspector_20 : TcoInspectors.TcoAnalogueInspector(THISSTRUCT);
    END_STRUCT
END_TYPE

// ---- Technology/Data/TechnologyData.TcDUT
{attribute clr [Container(Layout.Tabs)]}
TYPE
    TechnologyData EXTENDS TcoEntityBase :
    STRUCT

        CU00x : CU00xTechnologicalData := (Parent := THISSTRUCT);
		CU010 : CU010TechnologicalData := (Parent := THISSTRUCT);
		CU020 : CU020TechnologicalData := (Parent := THISSTRUCT);
		CU030 : CU030TechnologicalData := (Parent := THISSTRUCT);
		CU040 : CU040TechnologicalData := (Parent := THISSTRUCT);
		CU050 : CU050TechnologicalData := (Parent := THISSTRUCT);
    END_STRUCT
END_TYPE

// ---- Technology/TechnologyComponents.TcDUT
{attribute wpf [Container(Layout.Tabs)]}
TYPE
    TechnologyComponents EXTENDS TcoCore.TcoStruct :
    STRUCT
		//*{attribute wpf [Container(Layout.Stack, "Carousel")]}
		Carousel : TcoElements.TcoCarousel(THISSTRUCT);	
	
      	{attribute wpf [Container(Layout.Stack,"PRESURE")]}
        {attribute addProperty Name "<#Presure OK#>"}
        AirPresureOk : TcoElements.TcoDi(THISSTRUCT);  
	
		{attribute wpf [Container(Layout.Stack,"ESTOPS")]}
        {attribute addProperty Name "<#Emergency Stop#>"}
        EmergencyStop : TcoEmergencyStop(THISSTRUCT);

		{attribute wpf [Container(Layout.Stack,"CONTROL VOLTAGE")]}
        {attribute addProperty Name "<#Global control voltage#>"}
        GlobalControlVoltage : TcoControlVoltage(THISSTRUCT);
		

        {attribute addProperty Name "<#Local control voltage#>"}
        LocalControlVoltage : TcoControlVoltage(THISSTRUCT);
		

        {attribute addProperty Name "<#Local door voltage#>"}
        LocalDoorVoltage : TcoControlVoltage(THISSTRUCT);
		
		
		{attribute wpf [Container(Layout.Stack,"CONTROLS")]}
        {attribute addProperty Name "<#Control Buttons#>"}
        ControlButtons : TcoControlButtons(THISSTRUCT);
		
		{attribute addProperty Name "<#Virtual Control Buttons#>"}
        VirtualControlButtons : TcoControlButtons(THISSTRUCT);
		
		{attribute addProperty Name "<#Virtual Buttons#>"}
        VirtualButtons : VirtualButtons;
		
        {attribute addProperty Name "<#Mode key#>"}
        ModeKey : TcoKeyMode(THISSTRUCT);
		
		{attribute addProperty Name "<#Normal/Service key#>"}
        NormalServiceKey : TcoKeyNormalService(THISSTRUCT);
		
		{attribute wpf [Container(Layout.Stack,"DOORS")]}
		{attribute addProperty Name "<#Standard door#>"}
        StandardDoor : TcoStandardDoor(THISSTRUCT);

		{attribute addProperty Name "<#Basic door#>"}
        BasicDoor : TcoBasicDoor(THISSTRUCT);

		
		{attribute wpf [Container(Layout.Stack,"DOORCIRUITS AND ZONES")]}
		{attribute addProperty Name "<#Door circuit#>"}
        DoorCicuit : TcoDoorCircuit(THISSTRUCT);

		
		{attribute addProperty Name "<#Zone#>"}
        Zone : TcoControlledZone(THISSTRUCT);



    END_STRUCT
END_TYPE

// ---- Abstractions/Components/MtsFeeding/Blisters/Pls/TcoPlsPaletizator.TcPOU
FUNCTION_BLOCK TcoPlsPaletizator EXTENDS TcoCore.TcoComponent
VAR_INPUT
    inSafeCondition : BOOL;
	inSafeConditionErrorMsg : STRING; ///use this to insert specific safe condition message, otherwise a generic one is used
    inDoorOpen : BOOL;
END_VAR

VAR_OUTPUT
END_VAR
VAR
    {attribute addProperty Name "<#Config#>"}
    _config : TcoPlsPaletizator_Config_v_1_x_x;
    {attribute addProperty Name "<#Status#>"}
    {attribute clr [ReadOnly()]}
    _status : TcoPlsPaletizator_Status_v_1_x_x;
    {attribute addProperty Name "<#Control#>"}
    _control : TcoPlsPaletizator_Control_v_1_x_x;

    {attribute addProperty Name "<#Components#>"}
    _components : TcoPlsPaletizator_Components := (Parent := THIS^);

    {attribute addProperty Name "<#Request new blister#>"}
    _feedNewBlisterTask : TcoFeedingSequenceTask(THIS^);
    {attribute addProperty Name "<#Request to unload blister#>"}
    _throwBlisterTask : TcoFeedingSequenceTask(THIS^);
    {attribute addProperty Name "<#Request outgoing buffer#>"}
    _hanldeOutBufferTask : TcoFeedingSequenceTask(THIS^);
    {attribute addProperty Name "<#Request home position#>"}
    _setToDefaultTask : TcoFeedingSequenceTask(THIS^);

    {attribute addProperty Name "<#Restore#>"}
    _restoreTask : TcoCore.TcoTask(THIS^);

    
	
	
    {attribute addProperty Name "<#Safety temporarily disabled#>"}
    _temporarilyDisableSafety : BOOL;


    
	

	//~
	_blinker : TcoBlinker(THIS^);
	restoreDone : BOOL;
	_setSequencesToStep : BOOL := FALSE;
	_safeConditionErrorMsg : STRING;
    _timerEntryEmpty : TON;
    _timerOutFull : TON;
    _timerDisableSafety : TON;
	//~
END_VAR

_status.SafeCondition := inSafeCondition;
IF inSafeConditionErrorMsg <> '' THEN
	_safeConditionErrorMsg := inSafeConditionErrorMsg;
ELSE
	_safeConditionErrorMsg := '<#Safety condition not met!#>';
END_IF

Context.Environment.Messaging.Suspend();
_status.EntryBufferEmpty := NOT Components.I3_PresentBlistersInBufferEmpty.Signal;
_status.BlisterReady := Components.I4_PresentBlisterInWorkingPos.Signal AND Components.P7_SupportEntryBlister.AtWork;
_status.OutBufferFull := Components.I8_OutBlistersBufferIsFull.Signal;
Context.Environment.Messaging.Resume();

IF _config.StepModeManagableFromOutside THEN
    IF _setSequencesToStep THEN
        _feedNewBlisterTask.SetStepMode();
        _throwBlisterTask.SetStepMode();
        _hanldeOutBufferTask.SetStepMode();
        _setToDefaultTask.SetStepMode();
    ELSE
        _feedNewBlisterTask.SetCyclicMode();
        _throwBlisterTask.SetCyclicMode();
        _hanldeOutBufferTask.SetCyclicMode();
        _setToDefaultTask.SetCyclicMode();
    END_IF
END_IF;

_feedNewBlisterTask.Enabled := NOT _throwBlisterTask.Busy;
IF (_feedNewBlisterTask.Execute()) THEN
    SequenceIncomingBlister(refSequenceTask := _feedNewBlisterTask);
END_IF;

_throwBlisterTask.Enabled := NOT _feedNewBlisterTask.Busy;
IF (_throwBlisterTask.Execute()) THEN
    SequenceOutgoingBlister(refSequenceTask := _throwBlisterTask);
END_IF;

_hanldeOutBufferTask.Enabled := TRUE;
IF (_hanldeOutBufferTask.Execute()) THEN
    SequenceOutgoingBuffer(refSequenceTask := _hanldeOutBufferTask);
END_IF;

_setToDefaultTask.Enabled := TRUE;
IF (_setToDefaultTask.Execute()) THEN
    SequenceResetToDefault(refSequenceTask := _setToDefaultTask);
END_IF;

//*************RESTORE********************

_restoreTask.Enabled := TRUE;

IF _restoreTask.Execute() THEN
    Restore();
    _restoreTask.DoneWhen(inCondition := TRUE);
END_IF

//****************************************

//********************SAFETY******************
_timerDisableSafety(IN := _temporarilyDisableSafety, PT := _config.TimeToDisableSafety);

THIS^.Messenger.OnCondition(inCondition := _temporarilyDisableSafety).Warning('<#SAFETY TEMPORARILY DISABLED!#>');

IF NOT _temporarilyDisableSafety THEN

    Components.P7_SupportEntryBlister
        .SuspendMoveWorkExpression( Components.P7_SupportEntryBlister.MoveWorkTask.Busy AND NOT inSafeCondition, CONCAT('P7 <#Movement blocked#>: ',_safeConditionErrorMsg));

    Components.P7_SupportEntryBlister
        .SuspendMoveHomeExpression(Components.P7_SupportEntryBlister.MoveHomeTask.Busy AND NOT inSafeCondition, CONCAT('P7 <#Movement blocked#>: ',_safeConditionErrorMsg));

    Components.P8_FixEntryBlisterSide
        .SuspendMoveWorkExpression(Components.P8_FixEntryBlisterSide.MoveWorkTask.Busy AND NOT inSafeCondition, CONCAT('P8 <#Movement blocked#>: ',_safeConditionErrorMsg));

    Components.P8_FixEntryBlisterSide
        .SuspendMoveHomeExpression(Components.P8_FixEntryBlisterSide.MoveHomeTask.Busy AND NOT inSafeCondition, CONCAT('P8 <#Movement blocked#>: ',_safeConditionErrorMsg));

    IF NOT _config.LockBlisterInPickPosInactive THEN
        Components.P9_LockEntryBlisterTop
            .SuspendMoveWorkExpression(Components.P9_LockEntryBlisterTop.MoveWorkTask.Busy AND NOT inSafeCondition, CONCAT('P9 <#Movement blocked#>: ',_safeConditionErrorMsg));

        Components.P9_LockEntryBlisterTop
            .SuspendMoveHomeExpression(Components.P9_LockEntryBlisterTop.MoveHomeTask.Busy AND NOT inSafeCondition, CONCAT('P9 <#Movement blocked#>: ',_safeConditionErrorMsg));
    END_IF;

    Components.P4_FeedEntryBlister
        .SuspendMoveWorkExpression(NOT Components.P7_SupportEntryBlister.AtHome, CONCAT('P4 <#Movement blocked#>: ','<#P7 is not in home position#>'));

    Components.P4_FeedEntryBlister
        .SuspendMoveHomeExpression(NOT Components.P6_VerticalSepareOutBlister.AtHome, CONCAT('P4 <#Movement blocked#>: ','<#P6 is not in home position#>'));

    Components.P4_FeedEntryBlister
        .SuspendMoveHomeExpression(NOT Components.P5_HorizontalSepareOutBlisters.AtHome, CONCAT('P4 <#Movement blocked#>: ','<#P5 is not in home position#>'));

    Components.P4_FeedEntryBlister
        .SuspendMoveHomeExpression(Components.I7_OutBlistersIsAboveOutBuffer.Signal, CONCAT('P4 <#Movement blocked#>: ','<#empty blister is not unloaded#>'));

    Components.P7_SupportEntryBlister
        .SuspendMoveWorkExpression(NOT Components.P4_FeedEntryBlister.AtHome, CONCAT('P4 <#Movement blocked#>: ','<#P4 is not in home position#>'));

END_IF;

IF _timerDisableSafety.Q THEN
    _temporarilyDisableSafety := FALSE;
END_IF

PROPERTY Components : REFERENCE TO TcoPlsPaletizator_Components
GET
Components ref=_components;
END_GET
END_PROPERTY

(*~
	<docu>
		<summary>
			Gets the configuration of the MTS Pls feeder. 					
		</summary>			
	</docu>	
~*)
PROPERTY Config : REFERENCE TO TcoPlsPaletizator_Config_v_1_x_x
GET
Config REF= _config;
END_GET
END_PROPERTY

METHOD PUBLIC DefaultSignalisation
VAR_INPUT
END_VAR
Components.Q1_AttentionSignalisationR.Reset();
Components.Q2_AttentionSignalisationG.Reset();
Components.Q3_AttentionSignalisationB.Reset();

_blinker(inOffTime:=_config.BlinkTime,inOnTime:=_config.BlinkTime);
_timerEntryEmpty(in:= _status.EntryBufferEmpty,Pt:=_config.InfoTime);
_timerOutFull(in:=  _status.OutBufferFull ,Pt:=_config.InfoTime);
IF NOT inDoorOpen  
	AND NOT _timerEntryEmpty.Q
	AND NOT _timerOutFull.q THEN
	Components.Q2_AttentionSignalisationG.Set();
ELSIF  _blinker.IsOn THEN
	IF inDoorOpen AND 
		(
		THIS^._feedNewBlisterTask.Busy
		OR
		THIS^._throwBlisterTask.Busy
		OR
		THIS^._hanldeOutBufferTask.Busy )THEN
		Messenger.Warning('<#Waiting for palletizer service - Close the door!#>');
		Components.Q1_AttentionSignalisationR.Set();
		Components.Q2_AttentionSignalisationG.Set();
	ELSIF _timerEntryEmpty.Q
		THEN
		Components.Q1_AttentionSignalisationR.Set();
		Components.Q2_AttentionSignalisationG.Set();
	ELSIF _timerOutFull.Q
		THEN
		
		Components.Q1_AttentionSignalisationR.Set();
		Components.Q2_AttentionSignalisationG.Set();

//	ELSIF NOT _status.OutBufferFull
//		AND _status.EntryBufferEmpty 
//		AND NOT _status.BlisterReady THEN	
//		Components.Q1_AttentionSignalisationR.Set();
//	ELSIF  _status.OutBufferFull  THEN
//		Components.Q1_AttentionSignalisationR.Set();	
	
	END_IF;


	
END_IF;
END_METHOD

METHOD PUBLIC FeedNewBlister : TcoCore.ITcoTaskStatus

FeedNewBlister := _feedNewBlisterTask.Invoke();
END_METHOD

PROPERTY FeedNewBlisterTask : REFERENCE TO TcoFeedingSequenceTask
GET
FeedNewBlisterTask ref=_feedNewBlisterTask;
END_GET
END_PROPERTY

PROPERTY HandleOutBufferTask : REFERENCE TO TcoFeedingSequenceTask
GET
HandleOutBufferTask ref=_hanldeOutBufferTask;
END_GET
END_PROPERTY

PROPERTY OutBufferFull : bool
GET
OutBufferFull:=_status.OutBufferFull;
END_GET
END_PROPERTY

PROPERTY ReadyToUnloadComponent : bool
GET
ReadyToUnloadComponent:=_status.BlisterReady;
END_GET
END_PROPERTY

(*~
	<docu>
		<summary>
			Restores this instance to the Ready state. Can be called explicitly or from within one of the restore mechanisms.	
		</summary>			
	</docu>	
~*)
METHOD  Restore : ITcoRestorable
_hanldeOutBufferTask.Restore();
_feedNewBlisterTask.Restore();
_throwBlisterTask.Restore();
_setToDefaultTask.Restore();
_messenger.UnPin();
END_METHOD

METHOD PRIVATE SequenceIncomingBlister
VAR_INPUT
	refSequenceTask : REFERENCE TO TcoFeedingSequenceTask;
	
	
END_VAR

VAR
    seq    : REFERENCE TO TcoCore.TcoSequence;


END_VAR
seq REF= refSequenceTask.Sequence;
refSequenceTask(inoStatus:=_status,inoConfig:=_config);


seq.Open();
seq.Observer := refSequenceTask.Observer;



		



//***************************************************************************************************     
IF seq.Step(0,TRUE,'<#INITIAL SAFETY CHECK#>') THEN   
	     
	IF _status.SafeCondition THEN
    	seq.CompleteStep();
	ELSE
		Messenger.Warning(_safeConditionErrorMsg);
	END_IF;
END_IF        
//***************************************************************************************************     

 
//***************************************************************************************************     
IF seq.Step(10,TRUE,'<#CHECKING INCOMING BLISTERS#>') THEN   
    Messenger.Warning('<#BLISTER FEEDER EMPTY. REFILL INPUT BLISTERS!#>');
    seq.StepCompleteWhen(Components.I3_PresentBlistersInBufferEmpty.IsTrue);
END_IF      
//***************************************************************************************************     


        
//***************************************************************************************************     
IF seq.Step(20,TRUE,'<#ENTRY BLISTER SEPARATION#> - <#EXTENDING VERTICAL CYLINDERS#> P1, P2') THEN   

    seq.StepCompleteWhen(
        THIS^.Components.P1_VerticalSepareEntryBlisters.MoveToWork().Done AND
        THIS^.Components.P2_VerticalSepareEntryBlisters.MoveToWork().Done);

END_IF      
//***************************************************************************************************     


//***************************************************************************************************     
IF seq.Step(30,TRUE,'<#ENTRY BLISTER SEPARATION#> - <#RETRACTING CYLINDER#> P3') THEN   

    seq.StepCompleteWhen(
        THIS^.Components.P3_HorizontalSepareEntryBlisters.MoveToHome().Done);

END_IF    
//***************************************************************************************************     


//***************************************************************************************************     
IF seq.Step(40,TRUE,'<#ENTRY BLISTER SEPARATION#> - <#RETRACTING CYLINDER#> P1') THEN   

    seq.StepCompleteWhen(
        THIS^.Components.P1_VerticalSepareEntryBlisters.MoveToHome().Done);

END_IF      
//***************************************************************************************************     

//***************************************************************************************************     
IF seq.Step(45,TRUE,'<#ENTRY BLISTER SEPARATION#> - <#EXTENDING CYLINDER#> P2') THEN   

    seq.StepCompleteWhen(
        THIS^.Components.P2_VerticalSepareEntryBlisters.MoveToWork().Done);

END_IF       
//***************************************************************************************************     


//***************************************************************************************************     
IF seq.Step(50,TRUE,'<#ENTRY BLISTER SEPARATION#> - <#EXTENDING CYLINDERS#> P3, P10') THEN   

    seq.StepCompleteWhen(
        THIS^.Components.P3_HorizontalSepareEntryBlisters.MoveToWork().Done AND
        (Components.P10_HoldEntrySepareOutBlister.MoveToWork().Done OR _config.SepareBlistersAtEntryInactive));

END_IF       
//***************************************************************************************************     

//***************************************************************************************************     
IF seq.Step(60,TRUE,'<#ENTRY BLISTER SEPARATION#> - <#RETRACTING CYLINDERS#> P1, P2') THEN   

    seq.StepCompleteWhen(
        THIS^.Components.P1_VerticalSepareEntryBlisters.MoveToHome().Done AND
        THIS^.Components.P2_VerticalSepareEntryBlisters.MoveToHome().Done); 
					
END_IF       
//***************************************************************************************************     

//***************************************************************************************************     
IF seq.Step(65,NOT _config.SepareBlistersAtEntryInactive,'<#ENTRY BLISTER SEPARATION#> - <#RETRACTING CYLINDER#> P10') THEN   

    seq.StepCompleteWhen(
        Components.P10_HoldEntrySepareOutBlister.MoveToHome().Done);

END_IF       
//***************************************************************************************************     

//***************************************************************************************************   
IF seq.Step(70,TRUE,'<#CHECKING IF BLISTERS ARE SEPARATED#>') THEN   

    seq.StepCompleteWhen(
        THIS^.Components.I1_PresentBlisterEntry.IsTrue AND
        THIS^.Components.I2_PresentBlisterEntryEmptySpace.IsTrue);
		
	 Messenger.Error('I1, I2 <#FEEDER EMPTY, REFILL BLISTERS!#>');

END_IF    
//***************************************************************************************************     


//***************************************************************************************************     
IF seq.Step(80,TRUE,'<#ENTRY BLISTER HANDLING#> - <#RETRACTING SIDE CLAMP#> P8') THEN   

    seq.StepCompleteWhen(
        THIS^.Components.P8_FixEntryBlisterSide.MoveToHome().Done);

END_IF   
//***************************************************************************************************     

//***************************************************************************************************     
IF seq.Step(85,TRUE,'<#ENTRY BLISTER HANDLING#> - <#WAITING FOR TRANSFER TO WORK POSITION#> P4, I1') THEN   

    seq.StepCompleteWhen(
        THIS^.Components.P4_FeedEntryBlister.MoveToWork().Done AND
        Components.i4_PresentBlisterInWorkingPos.IsTrue);

END_IF  
//***************************************************************************************************     


//***************************************************************************************************     
IF seq.Step(90,TRUE,'<#ENTRY BLISTER HANDLING#> - <#CLAMPING BLISTER FROM THE SIDE#> P8') THEN   

    seq.StepCompleteWhen(
        THIS^.Components.P8_FixEntryBlisterSide.MoveToWork().Done);

END_IF   
//***************************************************************************************************     



//***************************************************************************************************     
IF seq.Step(100,TRUE,'<#ENTRY BLISTER HANDLING#> - <#MOVE TO PICK POSITION#> P6') THEN   

   IF THIS^.Components.P6_VerticalSepareOutBlister.AtHome THEN
	    seq.CompleteStep();
	ELSE
		Components.P6_VerticalSepareOutBlister.Messenger.Error(
            'P6 <#OUTPUT LIFT NOT IN UPPER POSITION!#>');
	END_IF

END_IF       
//***************************************************************************************************   

//***************************************************************************************************     
IF seq.Step(110,TRUE,'<#ENTRY BLISTER HANDLING#> - <#RETRACTING FEED#> P4') THEN   

	seq.StepCompleteWhen(
        THIS^.Components.P4_FeedEntryBlister.MoveToHome().Done);
	
END_IF 
//***************************************************************************************************   


//***************************************************************************************************     
IF seq.Step(120,TRUE,'<#ENTRY BLISTER HANDLING#> - <#LOWERING SUPPORT TRAY#> P7, P9') THEN   

    seq.StepCompleteWhen(
        THIS^.Components.P7_SupportEntryBlister.MoveToWork().Done AND
        (THIS^.Components.P9_LockEntryBlisterTop.MoveToHome().Done OR
         _config.LockBlisterInPickPosInactive));

END_IF       
//***************************************************************************************************   




IF (seq.Step(
    inStepID := seq.RESTORE_STEP_ID,
    inEnabled := TRUE,
    inStepDescription := '<#SEQUENCE COMPLETE#>')) THEN

    //--------------------------------------------------------	
    refSequenceTask.DoneWhen(TRUE);
    seq.CompleteSequence();
    //--------------------------------------------------------			

END_IF;


IF refSequenceTask.HandleTaskError() THEN
	//here we can decide what to do
	//	refSequenceTask.Restore();
	_feedNewBlisterTask.Restore();
END_IF



seq.Close();
END_METHOD

METHOD PRIVATE SequenceOutgoingBlister
VAR_INPUT
	refSequenceTask : REFERENCE TO TcoFeedingSequenceTask;
END_VAR

VAR
    seq    : REFERENCE TO TcoCore.TcoSequence;
END_VAR

VAR_INST
	_timer : TON;
END_VAR
seq REF= refSequenceTask.Sequence;
refSequenceTask(inoStatus:=_status,inoConfig:=_config);

seq.Open();
seq.Observer := refSequenceTask.Observer;



		



//***************************************************************************************************     
IF seq.Step(0,TRUE,'<#INITIAL SAFETY CHECK#>') THEN   
	IF _status.SafeCondition THEN
    	seq.CompleteStep();
	ELSE
		Messenger.Warning(_safeConditionErrorMsg);
	END_IF;
END_IF        
//***************************************************************************************************     

IF seq.Step(10,TRUE,'<#SEPARATING OUTGOING BLISTER#> - <#RELEASING BLISTER#> P9') THEN   

    seq.StepCompleteWhen(
        (THIS^.Components.P9_LockEntryBlisterTop.MoveToWork().Done OR
         _config.LockBlisterInPickPosInactive) AND
        THIS^.Components.P8_FixEntryBlisterSide.MoveToHome().Done);

END_IF  
//***************************************************************************************************   


//***************************************************************************************************     
IF seq.Step(20,TRUE,'<#SEPARATING OUTGOING BLISTER#> - <#LOWERING SUPPORT#> P7') THEN   

    seq.StepCompleteWhen(
        THIS^.Components.P7_SupportEntryBlister.MoveToHome().Done);

END_IF     
//***************************************************************************************************   



//***************************************************************************************************     
IF seq.Step(30,TRUE,'<#SEPARATING OUTGOING BLISTER#> - <#CHECKING BLISTER IN OUTPUT TRAY#> I5') THEN   
	IF seq.IsFreshState THEN
		_timer(IN:=FALSE);
	END_IF

	_timer(IN:=THIS^.Components.I5_OutBlistersIsThrowedCorrectly.Signal,
        PT:=_config.StabilisationTime);
	
	IF _timer.Q THEN
		seq.CompleteStep();
	ELSIF Components.P4_FeedEntryBlister.AtHome AND
       NOT THIS^.Components.I5_OutBlistersIsThrowedCorrectly.Signal THEN

		seq.StepCompleteWhen(
            seq.CurrentStep.Duration > _config.StabilisationTime);
	END_IF
	
END_IF    
//***************************************************************************************************   



IF (seq.Step(
    inStepID := seq.RESTORE_STEP_ID,
    inEnabled := TRUE,
    inStepDescription := '<#SEQUENCE COMPLETE#>')) THEN

    //--------------------------------------------------------	
    refSequenceTask.DoneWhen(TRUE);
    seq.CompleteSequence();
    //--------------------------------------------------------			

END_IF;


IF refSequenceTask.HandleTaskError() THEN
	//here we can decide what to do
	//	refSequenceTask.Restore();
	_throwBlisterTask.Restore();


END_IF


seq.Close();
END_METHOD

METHOD PRIVATE SequenceOutgoingBuffer
VAR_INPUT
	refSequenceTask : REFERENCE TO TcoFeedingSequenceTask;
	
	
END_VAR

VAR
    seq    : REFERENCE TO TcoCore.TcoSequence;

END_VAR

VAR_INST
	_timer:ton;
	
END_VAR
seq REF= refSequenceTask.Sequence;
refSequenceTask(inoStatus:=_status,inoConfig:=_config);

seq.Open();
seq.Observer := refSequenceTask.Observer;



		



//***************************************************************************************************     
IF seq.Step(0,TRUE,'<#INITIAL SAFETY CHECK#>') THEN   
	IF _status.SafeCondition THEN
    	seq.CompleteStep();
	ELSE
		Messenger.Warning(_safeConditionErrorMsg);
	END_IF;
END_IF         
//***************************************************************************************************     



//***************************************************************************************************     
IF seq.Step(10,TRUE,'<#OUTGOING BUFFER#> - <#CHECKING FOR BLISTER ABOVE THE BUFFER#> I7') THEN   

	IF seq.IsFreshState THEN
		_timer(IN:=FALSE);
	END_IF

	_timer(
        IN:=(*NOT THIS^.Components.I5_OutBlistersIsThrowedCorrectly.Signal AND*)
            Components.I7_OutBlistersIsAboveOutBuffer.Signal,
        PT:=_config.StabilisationTime);
	
    seq.StepCompleteWhen(_timer.Q);

END_IF        
//***************************************************************************************************   


//***************************************************************************************************     
IF seq.Step(20,TRUE,'<#OUTGOING BUFFER#> - <#CHECKING BLISTER COUNT#> I8') THEN   

	Messenger.Warning('<#FEEDER FULL, PLEASE REMOVE EMPTY BLISTERS!#>');

    seq.StepCompleteWhen(
        THIS^.Components.I8_OutBlistersBufferIsFull.IsFalse);

END_IF        
//***************************************************************************************************   


//***************************************************************************************************     
IF seq.Step(30,TRUE,'<#OUTGOING BUFFER#> - <#MOVING TRAYS ABOVE THE BLISTER#> P6') THEN   

	THIS^.Components.P6_VerticalSepareOutBlister.MoveToWork();

	IF Components.I6_OutBlistersLisftSignal.Signal THEN
	
		THIS^.Components.P6_VerticalSepareOutBlister.MoveWorkTask.Abort();
	    seq.StepCompleteWhen(TRUE);

	END_IF;
		
END_IF        
//***************************************************************************************************   


//***************************************************************************************************     
IF seq.Step(40,TRUE,'<#OUTGOING BUFFER#> - <#MOVING CYLINDER TO WORK POSITION#> P5') THEN   

	seq.StepCompleteWhen(
        Components.P5_HorizontalSepareOutBlisters.MoveToWork().Done);
		
END_IF        
//***************************************************************************************************   


//***************************************************************************************************     
IF seq.Step(45,TRUE,'<#OUTGOING BUFFER#> - <#HOMING CYLINDER#> P6') THEN   

	seq.StepCompleteWhen(THIS^.Components.P6_VerticalSepareOutBlister.MoveToHome().Done);
		
END_IF        
//***************************************************************************************************   


//***************************************************************************************************     
IF seq.Step(50,TRUE,'<#OUTGOING BUFFER#> - <#HOMING CYLINDER#> P5') THEN   

	seq.StepCompleteWhen(Components.P5_HorizontalSepareOutBlisters.MoveToHome().Done);
		
END_IF
//***************************************************************************************************   



IF (seq.Step(
    inStepID := seq.RESTORE_STEP_ID,
    inEnabled := TRUE,
    inStepDescription := '<#SEQUENCE COMPLETE#>')) THEN

    //--------------------------------------------------------	
    refSequenceTask.DoneWhen(TRUE);
    seq.CompleteSequence();
    //--------------------------------------------------------			

END_IF;


IF refSequenceTask.HandleTaskError() THEN
	//here we can decide what to do
	//refSequenceTask.Restore();
	_hanldeOutBufferTask.Restore();
END_IF


seq.Close();
END_METHOD

METHOD PRIVATE SequenceResetToDefault
VAR_INPUT
	refSequenceTask : REFERENCE TO TcoFeedingSequenceTask;
	
	
END_VAR

VAR
    seq    : REFERENCE TO TcoCore.TcoSequence;

END_VAR

VAR_INST
	_timer:ton;
	
END_VAR
seq REF= refSequenceTask.Sequence;
refSequenceTask(inoStatus:=_status,inoConfig:=_config);
seq.Open();
seq.Observer := refSequenceTask.Observer;



		



//***************************************************************************************************     
IF seq.Step(0,TRUE,'<#INITIAL SAFETY CHECK#>') THEN   
	IF _status.SafeCondition THEN
    	seq.CompleteStep();
	ELSE
		Messenger.Warning(_safeConditionErrorMsg);
	END_IF;
END_IF      
//***************************************************************************************************     



//***************************************************************************************************     
IF seq.Step(10,TRUE,'<#HOME POSITION#> - <#EXTENDING SEPARATOR CLAMPS#> P3') THEN   

    seq.StepCompleteWhen(
        Components.P3_HorizontalSepareEntryBlisters.MoveToWork().Done);

END_IF        
//***************************************************************************************************   


//***************************************************************************************************     
IF seq.Step(20,NOT _config.SepareBlistersAtEntryInactive,'<#HOME POSITION#> - <#RETRACTING CYLINDER#> P10') THEN   

    seq.StepCompleteWhen(
        Components.P10_HoldEntrySepareOutBlister.MoveToHome().Done);

END_IF        
//***************************************************************************************************   


//***************************************************************************************************     
IF seq.Step(30,TRUE,'<#HOME POSITION#> - <#LIFTING ENTRY BLISTERS#> P1, P2') THEN   

    seq.StepCompleteWhen(
        Components.P1_VerticalSepareEntryBlisters.MoveToHome().Done AND_THEN
        Components.P2_VerticalSepareEntryBlisters.MoveToHome().Done);

END_IF        
//***************************************************************************************************   


//***************************************************************************************************     
IF seq.Step(40,TRUE,'<#HOME POSITION#> - <#RETRACTING OUTPUT BLISTER CLAMPS#> P5') THEN   

	seq.StepCompleteWhen(
        Components.P5_HorizontalSepareOutBlisters.MoveToHome().Done);
		
END_IF        
//***************************************************************************************************   


//***************************************************************************************************     
IF seq.Step(50,TRUE,'<#HOME POSITION#> - <#RETRACTING OUTPUT BLISTER LIFT#> P6') THEN   

	seq.StepCompleteWhen(
        Components.P6_VerticalSepareOutBlister.MoveToHome().Done);
		
END_IF        
//***************************************************************************************************   


//***************************************************************************************************     
IF seq.Step(60,TRUE,'<#HOME POSITION#> - <#RETRACTING FEEDER#> P4') THEN   

	seq.StepCompleteWhen(
        Components.P4_FeedEntryBlister.MoveToHome().Done);
		
END_IF        
//***************************************************************************************************   


//***************************************************************************************************     
IF seq.Step(70,Components.I4_PresentBlisterInWorkingPos.Signal AND 
				Components.P8_FixEntryBlisterSide.AtWork,'<#HOME POSITION#> - <#LIFTING BLISTER SUPPORT#> P7, P9') THEN   

    seq.StepCompleteWhen(
        THIS^.Components.P7_SupportEntryBlister.MoveToWork().Done AND
        (THIS^.Components.P9_LockEntryBlisterTop.MoveToHome().Done OR
         _config.LockBlisterInPickPosInactive));

END_IF        
//***************************************************************************************************   


IF (seq.Step(inStepID := seq.RESTORE_STEP_ID,
    inEnabled := TRUE,
    inStepDescription := '<#SEQUENCE COMPLETE#>')) THEN
    //--------------------------------------------------------	
    refSequenceTask.DoneWhen(TRUE);
    seq.CompleteSequence();
    //--------------------------------------------------------			

END_IF;



IF refSequenceTask.HandleTaskError() THEN
	
	//here we can decide what to do
	//	refSequenceTask.Restore();

END_IF

seq.Close();
END_METHOD

(*~
	<docu>
		<summary>
		    Custom service (manual, maintenance) logic.
			This method must be implemented in derived class.
		</summary>			
	</docu>	
~*)
METHOD PROTECTED  ServiceMode
_components.Q3_AttentionSignalisationB.Service();
_components.Q2_AttentionSignalisationG.Service();
_components.Q1_AttentionSignalisationR.Service();
_components.P1_VerticalSepareEntryBlisters.Service();
_components.P2_VerticalSepareEntryBlisters.Service();
_components.P3_HorizontalSepareEntryBlisters.Service();
_components.P4_FeedEntryBlister.Service();
_components.P5_HorizontalSepareOutBlisters.Service();
_components.P6_VerticalSepareOutBlister.Service();
_components.P7_SupportEntryBlister.Service();
_components.P8_FixEntryBlisterSide.Service();
_components.P9_LockEntryBlisterTop.Service();
_components.P10_HoldEntrySepareOutBlister.Service();
END_METHOD

PROPERTY PUBLIC SetSequencesToStep : bool
GET
SetSequencesToStep:=_setSequencesToStep;
END_GET
SET
_setSequencesToStep:=SetSequencesToStep;
END_SET
END_PROPERTY

METHOD PUBLIC SetToDefault : TcoCore.ITcoTaskStatus
SetToDefault := _setToDefaultTask.Invoke();
END_METHOD

PROPERTY SetToDefaultTask : REFERENCE TO TcoFeedingSequenceTask
GET
SetToDefaultTask ref=_setToDefaultTask;
END_GET
END_PROPERTY

(*~
	<docu>
		<summary>
			Gets the status of the MTS Pls feeder. 					
		</summary>			
	</docu>	
~*)
PROPERTY Status : REFERENCE TO TcoPlsPaletizator_Status_v_1_x_x
GET
Status REF= _status;
END_GET
END_PROPERTY

METHOD PUBLIC ThrowBlister : TcoCore.ITcoTaskStatus

ThrowBlister := _throwBlisterTask.Invoke();
END_METHOD

PROPERTY ThrowBlisterTask : REFERENCE TO TcoFeedingSequenceTask
GET
ThrowBlisterTask ref=_throwBlisterTask;
END_GET
END_PROPERTY

END_FUNCTION_BLOCK

// ---- Abstractions/CUBase/CUBase.TcPOU
{attribute addProperty ShortName ""}
FUNCTION_BLOCK ABSTRACT CUBase EXTENDS TcoCore.TcoObject IMPLEMENTS ICUBase

VAR
    _cuId        : eStations;
    _processData : ProcessDataManager(THIS^);
	_groupInspection : TcoInspectors.TcoInspectionGroup(THIS^);
	{attribute addProperty Name "<#STATUS INFO#>"}
    _statusInfo  : CUBaseStatusInfo := (Parent := THIS^);
	_operatorInfo : OperatorInfo := (Parent := THIS^);
	_settings  : CUBaseSettings := (Parent := THIS^);
	//~
	_toggle: TcoUtilities.TcoBlinker(THIS^);
	//~
	_recurringFails:CuBaseRecurringFailures:=(Parent:=THIS^);
	_productionPlaner:ProductionPlaner(THIS^);
	_internalData : REFERENCE TO InternalStorage;	
	
	{attribute clr [ReadOnly()]}
	{attribute clr [RenderIgnore()]}
	_readyForOperations : BOOL;
END_VAR

(*~
	<docu>
		<summary>
			Controls `automatic` mode of `CU00x`.
		</summary>
	</docu>
~*)
METHOD  Automat
VAR_INPUT
END_VAR
(*
	Enable condition to start `automatTask`.
	Modify according your needs.
	[! 
	THIS IS NOT SAFETY CONDITION. THE SAFETY OF PRESONNEL AND EQUIPMENT MUST BE ENSURED BY ADDITIONAL MEANS 
	TO COMPLY WITH REGULATIONS
	]
*)


AutomatTask.Task.Enabled :=  AutomatTask.Task.Busy  XOR
							(GroundTask.GroundDone AND NOT AutomatTask.Task.Busy AND THIS^.Technology.AllowAutomat(inCuId:=CuId));

(*
	Invokes `groundTask` from technology object.
*)

IF(Technology.AutomatAllTask.Execute()) THEN AutomatTask.Task.Invoke(); END_IF;

IF(Technology.ForceStepMode()) THEN
 	AutomatTask.ModeController.Mode := eSequencerMode.StepMode;
END_IF
END_METHOD

PROPERTY ABSTRACT AutomatTask : REFERENCE TO CUBaseAutomat
GET
END_GET
END_PROPERTY

PROPERTY  CreateEntityTask : TcoCore.ITcoTaskStatus
GET
CreateEntityTask := _processData._createTask;
END_GET
END_PROPERTY

PROPERTY CuId : eStations
GET
CuId := _cuId;
END_GET
SET
_cuId := CuId;
END_SET
END_PROPERTY

PROPERTY  DeleteEntityTask : TcoCore.ITcoTaskStatus
GET
DeleteEntityTask := _processData._deleteTask;
END_GET
END_PROPERTY

METHOD DoesBelong : BOOL
DoesBelong := THIS^.ProcessDataManager.Data.EntityHeader.NextStation = THIS^.CuId;
END_METHOD

METHOD EntityFlowCloseForOperations : TcoCore.ITcoTaskStatus
VAR_IN_OUT
	Header : CuHeader; 
END_VAR
THIS^.FlagCloseEntity(Header);
EntityFlowCloseForOperations := THIS^.ProcessDataManager.Update(ProcessDataManager.Data._EntityId);
END_METHOD

METHOD EntityFlowCreateNew : TcoCore.ITcoTaskStatus
VAR_INPUT
	EntityId : STRING(255);	
END_VAR
VAR_IN_OUT
	Header : CuHeader;
END_VAR
THIS^.FlagCreateNewEntity(EntityId, Header);
EntityFlowCreateNew := THIS^.ProcessDataManager.Create(EntityId);
END_METHOD

METHOD EntityFlowDiscard : TcoCore.ITcoTaskStatus
VAR_INPUT
	EntityId : STRING(255);	
END_VAR
VAR_IN_OUT	
	Header : CuHeader; 
END_VAR
THIS^.FlagThrowAwayEntity(Header);
EntityFlowDiscard := THIS^.ProcessDataManager.Update(EntityId);
END_METHOD

METHOD EntityFlowFinalize : TcoCore.ITcoTaskStatus
VAR_IN_OUT
	Header : CuHeader; 
END_VAR
THIS^.FlagFinishEntity(Header);
EntityFlowFinalize := THIS^.ProcessDataManager.Update(ProcessDataManager.Data._EntityId);
END_METHOD

METHOD EntityFlowOpenForOperations : TcoCore.ITcoTaskStatus
VAR_INPUT
	Identifier : STRING(255);	
END_VAR
VAR_IN_OUT
	Header : CuHeader;
END_VAR
EntityFlowOpenForOperations := THIS^.ProcessDataManager.Read(Identifier);
THIS^.FlagOpenEntity(Identifier, Header);
END_METHOD

PROPERTY  ExistEntityTask : TcoCore.ITcoTaskStatus
GET
ExistEntityTask := _processData._idExistsTask;
END_GET
END_PROPERTY

METHOD PRIVATE FlagCloseEntity : BOOL
VAR_IN_OUT
	Header : CuHeader; 
END_VAR
THIS^.ProcessDataManager.Data.EntityHeader.LastStation := THIS^.CuId;

IF(THIS^.ProcessDataManager.Data.EntityHeader.Results.Result = TcoInspectors.eOverallResult.Failed) THEN	
	THIS^.ProcessDataManager.Data.EntityHeader.NextStation := Header.NextOnFailed;
ELSIF(THIS^.ProcessDataManager.Data.EntityHeader.Results.Result = TcoInspectors.eOverallResult.Passed) THEN
	THIS^.ProcessDataManager.Data.EntityHeader.NextStation := Header.NextOnPassed;
ELSIF(THIS^.ProcessDataManager.Data.EntityHeader.Results.Result = TcoInspectors.eOverallResult.InProgress) THEN
	THIS^.ProcessDataManager.Data.EntityHeader.NextStation := Header.NextOnPassed;
END_IF

THIS^.ProcessDataManager.Data.EntityHeader.OpenOn := eStations.NONE;
Header.CycleTime := THIS^._statusInfo.CurrentCycleTime;
Header.CleanLoopTime := THIS^._statusInfo.CurrentCleanCycleTime;
Header.OperationsEnded := Context.RealTimeClock.NowLocal();
Header.Operator := _operatorInfo.UserName;
END_METHOD

METHOD PRIVATE FlagCreateNewEntity : BOOL
VAR_INPUT
	Identifier : STRING(255);	
END_VAR
VAR_IN_OUT
	Header : CuHeader;
END_VAR
THIS^.ProcessDataManager.Data.EntityHeader.Results.Result := TcoInspectors.eOverallResult.InProgress;
THIS^.ProcessDataManager.Data._EntityId := Identifier;
THIS^.ProcessDataManager.Data.EntityHeader.WasReset := FALSE;
END_METHOD

METHOD PRIVATE FlagFinishEntity : BOOL
VAR_IN_OUT
	Header : CuHeader; 
END_VAR
THIS^.ProcessDataManager.Data.EntityHeader.LastStation := THIS^.CuId;

IF(THIS^.ProcessDataManager.Data.EntityHeader.Results.Result = TcoInspectors.eOverallResult.InProgress) THEN
	THIS^.ProcessDataManager.Data.EntityHeader.Results.Result := TcoInspectors.eOverallResult.Passed;
END_IF

IF(THIS^.ProcessDataManager.Data.EntityHeader.Results.Result = TcoInspectors.eOverallResult.Failed) THEN	
	THIS^.ProcessDataManager.Data.EntityHeader.NextStation := Header.NextOnFailed;
ELSIF(THIS^.ProcessDataManager.Data.EntityHeader.Results.Result = TcoInspectors.eOverallResult.Passed) THEN
	THIS^.ProcessDataManager.Data.EntityHeader.NextStation := Header.NextOnPassed;
END_IF

THIS^.ProcessDataManager.Data.EntityHeader.OpenOn := eStations.NONE;

Header.CycleTime := THIS^._statusInfo.CurrentCycleTime;
Header.CleanLoopTime := THIS^._statusInfo.CurrentCleanCycleTime;
Header.OperationsEnded := Context.RealTimeClock.NowLocal();
Header.Operator := _operatorInfo.UserName;
END_METHOD

METHOD PRIVATE FlagOpenEntity : BOOL
VAR_INPUT
	Identifier : STRING(255);	
END_VAR
VAR_IN_OUT
	Header : CuHeader;
END_VAR
Header.Operator := _operatorInfo.UserName;
Header.OperationsStarted := Context.RealTimeClock.NowLocal();
THIS^.ProcessDataManager.Data.EntityHeader.Results.Result := TcoInspectors.eOverallResult.InProgress;
THIS^.ProcessDataManager.Data._EntityId := Identifier;
THIS^.ProcessDataManager.Data.EntityHeader.OpenOn := THIS^.CuId;
THIS^.ProcessDataManager.Data.EntityHeader.WasReset := FALSE;
END_METHOD

METHOD PRIVATE FlagThrowAwayEntity : BOOL
VAR_IN_OUT	
	CuHeader : CuHeader; 
END_VAR
IF(THIS^.ProcessDataManager.Data.EntityHeader.OpenOn <> eStations.NONE) THEN
	THIS^.ProcessDataManager.Data.EntityHeader.LastStation := THIS^.CuId;
	THIS^.ProcessDataManager.Data.EntityHeader.NextStation := CuHeader.NextOnFailed;
	THIS^.ProcessDataManager.Data.EntityHeader.Results.Result := TcoInspectors.eOverallResult.Failed;
	THIS^.ProcessDataManager.Data.EntityHeader.WasReset := TRUE;
END_IF;
END_METHOD

(*~
	<docu>
		<summary>
			Controls `ground` mode of `CU00x`.
		</summary>
	</docu>
~*)
METHOD Ground : BOOL
VAR_INPUT
END_VAR
(*
	Enable condition to start `groundTask`.
	Modify according your needs.
	[! 
	THIS IS NOT SAFETY CONDITION. THE SAFETY OF PRESONNEL AND EQUIPMENT MUST BE ENSURED BY ADDITIONAL MEANS 
	TO COMPLY WITH REGULATIONS
	]
*)

GroundTask.Task.Enabled :=  THIS^.Technology.AllowGround(inCuId:=CuId)  OR GroundTask.Task.Busy ;

(*
	Invokes `groundTask` from technology object.
*)


IF(Technology.GroundAllTask.Execute()) THEN GroundTask.Restore();GroundTask.Task.Invoke(); END_IF;


IF GroundTask.GroundDone AND GroundTask.Task.Execute() THEN GroundTask.Restore();GroundTask.Task.Invoke();END_IF;
END_METHOD

PROPERTY ABSTRACT GroundTask : REFERENCE TO CUBaseGround
GET
END_GET
END_PROPERTY

PROPERTY FINAL GroupInspection : REFERENCE TO TcoInspectionGroup
GET
GroupInspection REF= _groupInspection;
END_GET
END_PROPERTY

(*~
	<docu>
		<summary>
			Code to be called cylically when `CU00x` idle; no other mode is active.
		</summary>
	</docu>
~*)
METHOD Idle : BOOL
END_METHOD

METHOD InternalCloseEntity : BOOL
VAR_INPUT
	inCarrier : UINT;
	refStorage : REFERENCE TO InternalStorage;
END_VAR
VAR_IN_OUT
	inoHeader : CuHeader; 
END_VAR
VAR_INST
	_internalData : REFERENCE TO InternalStorage;	
END_VAR
THIS^.FlagCloseEntity(inoHeader);
_internalData REF= refStorage;
InternalCloseEntity := _internalData.SaveByCarrier(inCarrier, THIS^.ProcessDataManager.Data);
END_METHOD

METHOD InternalCreateNewEntity : BOOL
VAR_INPUT
	inCarrier : UINT;
	refStorage : REFERENCE TO InternalStorage;
END_VAR
VAR_IN_OUT
	inoHeader : CuHeader; 
END_VAR
VAR_INST
	_internalData : REFERENCE TO InternalStorage;	
END_VAR
THIS^.FlagCreateNewEntity(UINT_TO_STRING(inCarrier), inoHeader);
THIS^.ProcessDataManager.Data.EntityHeader.Carrier := UINT_TO_STRING(inCarrier);
_internalData REF= refStorage;
InternalCreateNewEntity := _internalData.SaveByCarrier(inCarrier, THIS^.ProcessDataManager.Data);
END_METHOD

METHOD InternalFinishEntity : BOOL
VAR_INPUT
	inCarrier : UINT;
	refStorage : REFERENCE TO InternalStorage;
END_VAR
VAR_IN_OUT
	inoHeader : CuHeader; 
END_VAR
VAR_INST
	_internalData : REFERENCE TO InternalStorage;	
END_VAR
THIS^.FlagFinishEntity(inoHeader);

_internalData REF= refStorage;
InternalFinishEntity := _internalData.SaveByCarrier(inCarrier, THIS^.ProcessDataManager.Data);
END_METHOD

METHOD InternalOpenEntity : BOOL
VAR_INPUT
	inCarrier : UINT;
	refStorage : REFERENCE TO InternalStorage;
END_VAR
VAR_IN_OUT
	inoHeader : CuHeader; 
END_VAR
VAR_INST
	_internalData : REFERENCE TO InternalStorage;	
END_VAR
_internalData REF= refStorage;
InternalOpenEntity := _internalData.GetByCarrier(inCarrier, THIS^.ProcessDataManager.Data);
THIS^.FlagOpenEntity(UINT_TO_STRING(inCarrier), inoHeader);
END_METHOD

METHOD InternalRetrieveEntity : BOOL
VAR_INPUT
	inCarrier : UINT;
	refStorage : REFERENCE TO InternalStorage;
END_VAR
VAR_INST
	_internalData : REFERENCE TO InternalStorage;	
END_VAR
_internalData REF= refStorage;
InternalRetrieveEntity := _internalData.GetByCarrier(inCarrier, THIS^.ProcessDataManager.Data);
END_METHOD

METHOD InternalThrowAwayEntity : BOOL
VAR_INPUT
	inCarrier : UINT;
	refStorage : REFERENCE TO InternalStorage;
END_VAR
VAR_IN_OUT
	inoHeader : CuHeader; 
END_VAR
VAR_INST
	_internalData : REFERENCE TO InternalStorage;	
END_VAR
THIS^.FlagThrowAwayEntity(inoHeader);
_internalData REF= refStorage;
InternalThrowAwayEntity := _internalData.SaveByCarrier(inCarrier, THIS^.ProcessDataManager.Data);
END_METHOD

(*~
	<docu>
		<summary>
			Controls `manual` mode of `CU00x`.
		</summary>
	</docu>
~*)
METHOD Manual : BOOL
VAR_INPUT
END_VAR
(*
	Enable condition to start `automatTask`.
	Modify according your needs.
	[! 
	THIS IS NOT SAFETY CONDITION. THE SAFETY OF PRESONNEL AND EQUIPMENT MUST BE ENSURED BY ADDITIONAL MEANS 
	TO COMPLY WITH REGULATIONS
	]
*)

ManualTask.Task.Enabled :=  THIS^.Technology.AllowManual(inCuId:=CuId)  OR ManualTask.Task.Busy;
END_METHOD

PROPERTY ABSTRACT ManualTask : REFERENCE TO TcoTaskedService
GET
END_GET
END_PROPERTY

PROPERTY FINAL ProcessDataManager : REFERENCE TO ProcessDataManager
GET
ProcessDataManager REF= _processData;
END_GET
END_PROPERTY

PROPERTY  ReadEntityTask : TcoCore.ITcoTaskStatus
GET
ReadEntityTask := _processData._readTask;
END_GET
END_PROPERTY

METHOD ReadyForOperations : BOOL
VAR_INPUT
END_VAR
ReadyForOperations := _readyForOperations;
END_METHOD

PROPERTY ABSTRACT RecoverTask : REFERENCE TO CUBaseRecover
GET
END_GET
END_PROPERTY

PROPERTY RecurringFails : REFERENCE TO CuBaseRecurringFailures
GET
RecurringFails REF= _recurringFails;
END_GET
END_PROPERTY

METHOD ResetReadyForOperations : BOOL
_readyForOperations := false;
END_METHOD

METHOD  RunOperations : BOOL
VAR_INPUT
	refGlobalTrigger:REFERENCE TO BOOL;
END_VAR
VAR
	_trrigger:REFERENCE TO BOOL;
END_VAR
_trrigger REF=refGlobalTrigger;
RunOperations := _trrigger;
END_METHOD

METHOD  SetReadyForOperations : BOOL
VAR_INPUT
END_VAR
_readyForOperations := TRUE;
END_METHOD

PROPERTY ABSTRACT StatusInfo : REFERENCE TO CUBaseStatusInfo
GET
END_GET
END_PROPERTY

PROPERTY ABSTRACT SuspendTask : REFERENCE TO CUBaseSuspend
GET
END_GET
END_PROPERTY

PROPERTY Technology : REFERENCE TO Technology
GET
VAR
    _technology : POINTER TO Technology;
END_VAR
IF __QUERYPOINTER(Parent, _technology) THEN // Check if _Parent is Station001
    Technology REF= _technology^;              // If the check is successful dereference a pointer. simlar to THIS^ or SUPER^
END_IF
END_GET
END_PROPERTY

PROPERTY PUBLIC ToggleBlinker : REFERENCE TO TcoUtilities.TcoBlinker
GET
ToggleBlinker ref= _toggle;
END_GET
END_PROPERTY

PROPERTY  UpdateEntityTask : TcoCore.ITcoTaskStatus
GET
UpdateEntityTask := _processData._updateTask;
END_GET
END_PROPERTY

METHOD UpdateInfo : BOOL
VAR_INPUT
END_VAR
_toggle(inOffTime:=T#500MS,inOnTime:=T#500MS);

IF AutomatTask.ClearCounterDataTask.Execute() THEN
	AutomatTask.ClearCounter();
	AutomatTask.ClearCounterDataTask.DoneWhen(TRUE);
END_IF

_statusInfo.State := eCUState.None;

IF _statusInfo.CurrentCleanCycleTime  >= _settings.WarningCycleTime
	AND _statusInfo.CurrentCleanCycleTime  < _settings.ErrorCycleTime THEN
	_statusInfo.State:= eCUState.HasWarning;
ELSIF _statusInfo.CurrentCleanCycleTime   >= _settings.ErrorCycleTime THEN
	_statusInfo.State := eCUState.HasError;
END_IF; 


IF _toggle.IsOff THEN
	_statusInfo.State := eCUState.None;
END_IF



IF AutomatTask.Task.Busy THEN

    _statusInfo.Mode                   := eCUMode.AutomatMode;
    _statusInfo.CurrentTaskDescription := '<#AUTOMAT#>';
    _statusInfo.CurrentCycleTime       := AutomatTask._SequenceElapsedTime;
	_statusInfo.CurrentCleanCycleTime  := T#0S;

	IF AutomatTask._startCleanCycleTime<>T#0S AND AutomatTask._stopCleanCycleTime=T#0S  THEN
		_statusInfo.CurrentCleanCycleTime  := AutomatTask._SequenceElapsedTime-AutomatTask._startCleanCycleTime;
	ELSIF AutomatTask._stopCleanCycleTime<>T#0S  THEN
		_statusInfo.CurrentCleanCycleTime  := AutomatTask._stopCleanCycleTime-AutomatTask._startCleanCycleTime;
	ELSE
		_statusInfo.CurrentCleanCycleTime :=AutomatTask._startCleanCycleTime;
	END_IF;
	
	_statusInfo.AverageCycleTime	   := AutomatTask.AverageCycleTime;
	_statusInfo.AverageCleanCycleTime  := AutomatTask.AverageCleanCycleTime;
    _statusInfo.CurrentUid             := AutomatTask.CurrentStep.ID;
    _statusInfo.CurrentOperation       := AutomatTask.CurrentStep.Description;
    _statusInfo.CurrentIsInStepMode    := AutomatTask._modeController._mode = eSequencerMode.StepMode;
ELSIF GroundTask.Task.Busy THEN
    _statusInfo.Mode := eCUMode.GroundMode;
	_statusInfo.CurrentTaskDescription := '<#GROUND#>';
    _statusInfo.CurrentCycleTime       := GroundTask._SequenceElapsedTime;
	_statusInfo.CurrentCleanCycleTime := T#0S;
	_statusInfo.AverageCycleTime	   := GroundTask.AverageCycleTime;
	_statusInfo.AverageCleanCycleTime  := T#0S;
    _statusInfo.CurrentUid             := GroundTask.CurrentStep.ID;
    _statusInfo.CurrentOperation       := GroundTask.CurrentStep.Description;
    _statusInfo.CurrentIsInStepMode    := GroundTask._modeController._mode = eSequencerMode.StepMode;
ELSIF THIS^.ManualTask.Busy THEN
    _statusInfo.Mode := eCUMode.ManualMode;
	_statusInfo.CurrentTaskDescription := '<#MANUAL#>';
	_statusInfo.State := eCUState.None;
	_statusInfo.CurrentIsInStepMode    := FALSE;

ELSIF THIS^.GroundTask.Task.Done THEN
	_statusInfo.CurrentTaskDescription := '<#READY TO START#>';
	_statusInfo.Mode := eCUMode.GroundModeDone;
	_statusInfo.CurrentCycleTime       := GroundTask._SequenceElapsedTime;
    _statusInfo.CurrentUid             := GroundTask.CurrentStep.ID;
    _statusInfo.CurrentOperation       := GroundTask.CurrentStep.Description;
    _statusInfo.CurrentIsInStepMode    := GroundTask._modeController._mode = eSequencerMode.StepMode;
	_statusInfo.State := eCUState.None;

ELSE
    _statusInfo.Mode := eCUMode.NoMode;	
	_statusInfo.CurrentTaskDescription := '<#IDLE#>';
	_statusInfo.CurrentCycleTime       := T#0S;
    _statusInfo.CurrentUid             := 0;
    _statusInfo.CurrentOperation       := '';
    _statusInfo.CurrentIsInStepMode    := FALSE;
	_statusInfo.State := eCUState.None;
END_IF
END_METHOD

END_FUNCTION_BLOCK

// ---- Technology/Data/InternalStorage.TcPOU
FUNCTION_BLOCK InternalStorage EXTENDS TcoCore.TcoObject 
VAR
	_data : ARRAY [0..9] OF ProcessData := [(Parent := THIS^), (Parent := THIS^), (Parent := THIS^), (Parent := THIS^), (Parent := THIS^),
                                        (Parent := THIS^), (Parent := THIS^), (Parent := THIS^), (Parent := THIS^), (Parent := THIS^)];
END_VAR
VAR CONSTANT
	_maxNumberOfCarriers : UINT := 10;
END_VAR

METHOD GetByCarrier : BOOL
VAR_INPUT
	inCarrier : UINT;
END_VAR
VAR_IN_OUT
	inoData : ProcessData;
END_VAR
IF(inCarrier >= 0 AND inCarrier < _maxNumberOfCarriers) THEN
	inoData := _data[inCarrier];
	GetByCarrier := TRUE;
	RETURN;	
END_IF

Messenger.Post(CONCAT('<#Requested carrier is out of range of internal storage. Max number of carriers is#> ', UINT_TO_STRING(_maxNumberOfCarriers)), eMessageCategory.ProgrammingError);
END_METHOD

METHOD SaveByCarrier : BOOL
VAR_INPUT
	inCarrier : UINT;
END_VAR
VAR_IN_OUT
	inoData : ProcessData;
END_VAR
IF(inCarrier >= 0 AND inCarrier < _maxNumberOfCarriers) THEN
	_data[inCarrier] := inoData;
	SaveByCarrier := TRUE;
	RETURN;	
END_IF

Messenger.Post(CONCAT('<#Requested carrier is out of range of internal storage. Max number of carriers is#> ', UINT_TO_STRING(_maxNumberOfCarriers)), eMessageCategory.ProgrammingError);
END_METHOD

END_FUNCTION_BLOCK

// ---- Technology/Technology.TcPOU
FUNCTION_BLOCK Technology EXTENDS TcoCore.TcoContext
VAR	
    _processSettings     : ProcessDataManager(THIS^);  			//a.k.a receipe
	_reworkSettings     : ProcessDataManager(THIS^);  			//a.k.a receipe for rework
    _technologySettings  : TechnologicalDataManager(THIS^);		//a.k.a machine settings
    _processTraceability : ProcessDataManager(THIS^);			//the same structure as process setting but filled with actual production data (measurements, inspection results, etc)
	//~
	_internalStorage : InternalStorage(THIS^);					//
	//~
	
	fbGetCurTaskIndex            : GETCURTASKINDEX;
	_notificationPanel      : NotificationPanel(THIS^);				//provide technology state signals to side baner in visualisation
    {attribute addProperty Name "<#AUTOMAT ALL#>"}
    _automatAllTask : TcoCore.TcoTask(THIS^);					// Commmand-like taks to execute automation mode on whole technology. Handled in controlled units.
    {attribute addProperty Name "<#GROUND ALL#>"}
    _groundAllTask : TcoCore.TcoTask(THIS^);	

	{attribute addProperty Name "<#_cu00x#>"}					
    _cu00x         : CU00x(THIS^);
		{attribute addProperty Name "<#_cu010#>"}					
    _cu010         : CU010(THIS^);
		{attribute addProperty Name "<#_cu020#>"}					
    _cu020         : CU020(THIS^);
		{attribute addProperty Name "<#_cu030#>"}					
    _cu030         : CU030(THIS^);
		{attribute addProperty Name "<#_cu040#>"}					
    _cu040        : CU040(THIS^);
			{attribute addProperty Name "<#_cu050#>"}					
    _cu050        : CU050(THIS^);
	
	{attribute addProperty Name "<#Technology Components#>"}	
	_components : TechnologyComponents:= (Parent := THIS^);

	{attribute addProperty Name "Device 1 (EtherCAT)"}
	Device_1 : TcoIo.TcoEthercatMasterDevice(THIS^);
	
	_setDummyConditionsSuffisient:BOOL;
	//~
	_dummyBlinker              : TcoUtilities.TcoBlinker(THIS^);
	//~
	_runOperations:BOOL;

	
END_VAR

METHOD AllowAutomat : BOOL
VAR_INPUT
	inCuId : eStations;
END_VAR

VAR
	retVal: BOOL;
END_VAR
retVal := FALSE;
IF inCuId = eStations.CU00x THEN
	 retVal := TRUE;// Components.Zone1.Status.State.AnyKeyManual AND Components.ControlVoltages.R1.GlobalControlVoltage.Signal;
END_IF;


AllowAutomat := retVal;
END_METHOD

METHOD AllowGround : BOOL
VAR_INPUT
	inCuId : eStations;
END_VAR

VAR
	retVal: BOOL;
END_VAR
retVal := FALSE;
IF inCuId = eStations.CU00x THEN
	 retVal := TRUE;// Components.Zone1.Status.State.AnyKeyManual AND Components.ControlVoltages.R1.GlobalControlVoltage.Signal;
END_IF;


AllowGround := retVal;
END_METHOD

METHOD AllowManual :  BOOL
VAR_INPUT
	inCuId : eStations;
END_VAR


VAR
	retVal: BOOL;
END_VAR
retVal := FALSE;
IF inCuId = eStations.CU00x THEN
	 retVal := TRUE;// Components.Zone1.Status.State.AnyKeyManual AND Components.ControlVoltages.R1.GlobalControlVoltage.Signal;
END_IF;


AllowManual := retVal;
END_METHOD

PROPERTY AutomatAllTask : REFERENCE TO TcoCore.TcoTask
GET
AutomatAllTask REF= _automatAllTask;
END_GET
END_PROPERTY

PROPERTY Components : REFERENCE TO TechnologyComponents
GET
Components REF= _components;
END_GET
END_PROPERTY

PROPERTY PUBLIC Cu00x : Reference to CU00x
GET
Cu00x REF=_cu00x;
END_GET
END_PROPERTY

METHOD ForceStepMode : BOOL
ForceStepMode := FALSE;
END_METHOD

PROPERTY GroundAllTask : REFERENCE TO TcoCore.TcoTask
GET
GroundAllTask REF= _groundAllTask;
END_GET
END_PROPERTY

METHOD InitializeComponents
VAR_INST
	DoNothing : BOOL;
	None : BOOL;
END_VAR

VAR
	controlVolage: BOOL;
	controlVoltageDoor: BOOL;
	estop: BOOL;
	presure: BOOL;
	locked: BOOL;
	lock: BOOL;
	opened: BOOL;
	closed: BOOL;
	
END_VAR
controlVolage:=FALSE;
controlVoltageDoor:=FALSE;
estop:=FALSE;
presure:=FALSE;

_components.VirtualControlButtons(
	refButtonRecover:= _components.VirtualButtons.StartButton, 
	refButtonSuspend:= _components.VirtualButtons.StopButton, 
	refButtonGround:= None , 
	refButtonAuto:= None, 
	refButtonRecoverLight:= _components.VirtualButtons.StartLight,
	refButtonSuspendLight:= _components.VirtualButtons.StopLight, 
	refButtonGroundLight:= DoNothing, 
	refButtonAutoLight:=  DoNothing);



//_dummyBlinker(inOffTime := T#10000MS, inOnTime := T#10000MS);
(*
closed:=GVL_iXlinker.EC1.EK1200.IA1_EL1809.Channel_8.Input;
locked:=GVL_iXlinker.EC1.EK1200.IA1_EL1809.Channel_9.Input;

IF _setDummyConditionsSuffisient THEN
	controlVolage:=TRUE;
	controlVoltageDoor:=TRUE;
	estop:=FALSE;
	presure:=TRUE;


END_IF;

_components.ModeKey(inoKeyState1:=GVL_iXlinker.EC1.EK1200.IA1_EL1809.Channel_1.Input ,
					inoKeyState2:=GVL_iXlinker.EC1.EK1200.IA1_EL1809.Channel_2.Input);
					
_components.NormalServiceKey(inoSignal:=GVL_iXlinker.EC1.EK1200.IA1_EL1809.Channel_3.Input);
					
_components.ControlButtons(
	inoButtonRecover:=GVL_iXlinker.EC1.EK1200.IA1_EL1809.Channel_4.Input  , 
	inoButtonSuspend:=GVL_iXlinker.EC1.EK1200.IA1_EL1809.Channel_5.Input  , 
	inoButtonGround:=GVL_iXlinker.EC1.EK1200.IA1_EL1809.Channel_6.Input , 
	inoButtonAuto:=GVL_iXlinker.EC1.EK1200.IA1_EL1809.Channel_7.Input, 
	inoButtonRecoverLight:=GVL_iXlinker.EC1.EK1200.QA1_EL2809.Channel_1.Output  , 
	inoButtonSuspendLight:=GVL_iXlinker.EC1.EK1200.QA1_EL2809.Channel_2.Output  , 
	inoButtonGroundLight:=GVL_iXlinker.EC1.EK1200.QA1_EL2809.Channel_3.Output  , 
	inoButtonAutoLight:= GVL_iXlinker.EC1.EK1200.QA1_EL2809.Channel_4.Output );
	

					

_components.GlobalControlVoltage(inoSignal := controlVolage);

_components.LocalControlVoltage(inoSignal := controlVolage);
_components.LocalDoorVoltage(inoSignal := controlVoltageDoor);

_components.EmergencyStop(inoSignal := estop);
_components.AirPresureOk(inoSignal:= presure);


_components.StandardDoor(inoIsLocked := locked,
    inoIsOpen := opened,
    inoLock :=lock);
	
	
_components.BasicDoor(inoIsClosed := closed,
     inoLock := lock);


_components.DoorCicuit();

_components.Zone(inDoorCircuit:=_components.DoorCicuit,
				inEstopActive:=_components.EmergencyStop.Signal,
				inAirPressureOK:= _components.AirPresureOk.Signal);
		
				
_components.Zone.Service();
*)
END_METHOD

METHOD InitializeComponentsOnce
VAR_INPUT
END_VAR
_components.DoorCicuit.Restore();
_components.Zone.Restore();



_components.DoorCicuit.AddDoors(inDoor:=_components.StandardDoor);
_components.DoorCicuit.AddDoors(inDoor:=_components.BasicDoor);
_components.DoorCicuit.AddGlobalVoltage(inVoltage:=_components.GlobalControlVoltage);
_components.DoorCicuit.AddLocalVoltage(inVoltage:=_components.LocalControlVoltage);
_components.DoorCicuit.AddLocalDoorsVoltage(inVoltage:=_components.LocalDoorVoltage);


_components.Zone.AddControlledUnit(inControlledUnit:=_cu00x);
_components.Zone.AddControlButtons(inControlButtons:=_components.ControlButtons);
_components.Zone.AddControlButtons(inControlButtons:=_components.VirtualControlButtons);

_components.Zone.AddKeyMode(inKeyMode:=_components.ModeKey);
_components.Zone.AddKeyNormalService(inKeyNormalService:=_components.NormalServiceKey);
END_METHOD

METHOD InitializeNotificationPanel
VAR
	//~
	icon : Icon;
	new : Icon;
	//~
END_VAR

VAR_INST
	//~
	tixonsOK : BOOL;
	tixonErrorTmr : TON;
	//~
END_VAR
Context.Environment.Messaging.Suspend();


{region "NOTIFICATION PANEL"}
_notificationPanel.Clear();


icon.Title := '<#Control Voltage#>';
icon.IconType := TO_STRING(eIconType.ControlVoltage);
icon.Signal := Components.GlobalControlVoltage.Signal;
_notificationPanel.addIcon(icon);
icon := new;

icon.Title := '<#Air Pressure#>';
icon.IconType := TO_STRING(eIconType.AirPressure);
icon.Signal := Components.AirPresureOk.Signal;
_notificationPanel.addIcon(icon);
icon := new;

icon.Title := '<#Emergency Stop#>';
icon.IconType := TO_STRING(eIconType.EmergencyStop);
icon.Signal := Components.EmergencyStop.Signal;
_notificationPanel.addIcon(icon);
icon := new;

icon.Title := '<#Safety door#>';
icon.IconType := TO_STRING(eIconType.SafetyDoor);
icon.Signal :=  Components.DoorCicuit.IsLocalDoorsVoltageOk;
_notificationPanel.addIcon(icon);
icon := new;

icon.Title := '<#Doors closed#>';
icon.IconType := TO_STRING(eIconType.DoorClosed);
icon.Signal := Components.DoorCicuit.IsClosed;
_notificationPanel.addIcon(icon);
icon := new;

icon.Title := '<#Doors Locked#>';
icon.IconType := TO_STRING(eIconType.DoorLocked);
icon.Signal := Components.DoorCicuit.IsLocked;
_notificationPanel.addIcon(icon);
icon := new;

icon.Title := '<#Automat Allowed#>';
icon.IconType := TO_STRING(eIconType.AutomatAllowed);
icon.Signal := Components.Zone.Status.State.AllKeysAuto;
_notificationPanel.addIcon(icon);
icon := new;

icon.Title := '<#Process Data Loaded#>';
icon.IconType := TO_STRING(eIconType.ProcessDataLoaded);
icon.Signal := ProcessSettings.Data._EntityId <> '';
_notificationPanel.addIcon(icon);
icon := new;

icon.Title := '<#Technology Data Loaded#>';
icon.IconType := TO_STRING(eIconType.TechnologyDataLoaded);  
icon.Signal := TechnologicalSettings.Data._EntityId <> '';
_notificationPanel.addIcon(icon);
icon := new;

icon.Title := '<#Manipulator#>';
icon.IconType := 'AxisArrow';  
/// Recommend to set a backing field in the affected CUs and accessing it through a property, because the below line WILL cause the the plc to crash in the first cycle!!! 
//icon.Signal := NOT _cu00x.Components.MultiAxis.Axis_1.AxisStatus.Error;
_notificationPanel.addIcon(icon);
icon := new;
	 
icon.Title := '<#Robots#>';
icon.IconType := TO_STRING(eIconType.Robot);  
icon.Signal :=  _cu00x.Components.KukaKrc4.Status.State.ExternalAutomatic AND NOT _cu00x.Components.KukaKrc4.Status.State.Error;
_notificationPanel.addIcon(icon);
icon := new;
	 

icon.Title := '<#Cameras#>';
icon.IconType := 'CameraOutline';  
icon.Signal := NOT _cu00x.Components.Cam.Status.SignalStatus.Error;
_notificationPanel.addIcon(icon);
icon := new;
	 
icon.Title := '<#Laser#>';
icon.IconType := 'Qrcode';
//icon.Signal := _cu00x.Components.KeyenceLaser.Status.MachineStatus.IsConnection;
_notificationPanel.addIcon(icon);
icon := new;

///Tixon Auto from project 2400620
//tixonErrorTmr(IN := (NOT _cu00x.Components.Tixon.Status.Ready AND NOT _cu00x.Components.Tixon.RequestSrcewTask.Busy) , PT := T#3S );
tixonsOK := NOT tixonErrorTmr.Q; 

icon.Title := 'TIXON';
icon.IconType := 'Bolt';  
icon.Signal := tixonsOK;
_notificationPanel.addIcon(icon);
icon := new;
	 
_notificationPanel();
{endregion}
 Context.Environment.Messaging.Resume();
END_METHOD

PROPERTY InternalStorage : REFERENCE TO InternalStorage
GET
InternalStorage REF= _internalStorage;
END_GET
END_PROPERTY

(*~
	<docu>
		<summary>
			Main method of the TcoContext. This is the entry point of any control logic that belongs to this context. 
			The call of this method is ensured by calling the <c>InstanceName.Run()</c> method, and it must not be called explicitly.
			This method is abstract, and it must be overridden in derived block.
		</summary>
	</docu>
~*)
METHOD PROTECTED Main
(*
	Context settings 
*)



// Messenger logger settings
_settings.Messaging.MessageDigestMethod := eMessageDigestMethod.CRC32;
_settings.Messaging.MessengerLoggingMethod := eMessengerLogMethod.OnEventRisen;


_components.DoorCicuit.Config.MaxDoors:=12;
_components.DoorCicuit.Config.MaxGlobalVoltage:=2;
_components.DoorCicuit.Config.MaxLocalVoltage:=2;
_components.DoorCicuit.Config.MaxLocalDoorsVoltage:=2;


_components.Zone.Config.MaxControlButtons:=2;
_components.Zone.Config.MaxControledUnits:=10;
_components.Zone.Config.MaxKeyMode:=2;
_components.Zone.Config.MaxKeyNormalService:=2;



THIS^.InitializeComponents();

fbGetCurTaskIndex();
IF _TaskInfo[fbGetCurTaskIndex.index].FirstCycle THEN
    // The code that you want to be executed at the first cycle of  PLC only 
	THIS^.InitializeComponentsOnce();
	
ELSE
	// RTC Synchronisation
	THIS^.RtcSynchronize(TRUE,  
					 '192.168.4.1.1.1',    // Provide AMS ID of the time source, leave blank if local. 
					 60);
END_IF

//notification panel
 Context.Environment.Messaging.Suspend();
			
 InitializeNotificationPanel();
			
 Context.Environment.Messaging.Resume();

(*
	
	Data managers

*)

_processSettings();
_reworkSettings();
_technologySettings();

(*

	Controlled units
	
*)

_cu00x();
_cu010();
_cu020();
_cu030();
_cu040();
_cu050();


_automatAllTask();
_groundAllTask();

//Device_1(	SyncUnits		:= ADR(		GVL_iXlinker.EC1.SyncUnits),
//			SyncUnitsSize	:= SIZEOF(	GVL_iXlinker.EC1.SyncUnits),
//			Inputs			:=			GVL_iXlinker.EC1.Inputs,
//			InfoData		:=			GVL_iXlinker.EC1.InfoData);
END_METHOD


(*~
	<docu>
		<summary>
			Called upon exit from the context. When overridden in derived class allows to execute an arbitrary logic after closing the context cycle.	
		</summary>			
	</docu>	
~*)METHOD PROTECTED OnExit
_automatAllTask.DoneWhen(TRUE);
_groundAllTask.DoneWhen(TRUE);
END_METHOD

PROPERTY ProcessSettings : REFERENCE TO ProcessDataManager
GET
ProcessSettings REF= _processSettings;
END_GET
END_PROPERTY

PROPERTY ReworkSettings : REFERENCE TO ProcessDataManager
GET
ReworkSettings REF= _reworkSettings;
END_GET
END_PROPERTY

PROPERTY RunOperations : REFERENCE TO BOOL
GET
RunOperations REF= _runOperations;
END_GET
END_PROPERTY

PROPERTY TechnologicalSettings : REFERENCE TO TechnologicalDataManager
GET
TechnologicalSettings REF= _technologySettings;
END_GET
END_PROPERTY

END_FUNCTION_BLOCK

// ---- Abstractions/Generic/NotificationPanel/NotificationPanel.TcPOU

    (*~
        <docu>
            <summary>Extendable notification panel</summary>
            <note>It is filled with icons in Technology.InitializeNotificationPanel() and updated on each cyle. 
Further extentions can be added in NotificationPanelView.xaml see SynologyNotificationView</note>
        </docu>
    ~*)
FUNCTION_BLOCK NotificationPanel EXTENDS TcoObject
VAR_INPUT
	(*~
		<docu>
			<summary>
				Time duration for toggle signal.
			</summary>
		</docu>
	~*)
	inBlinkPeriod : TIME := T#500MS;
END_VAR
VAR CONSTANT
	LAST_ICON_INDEX : INT := 19;
END_VAR

VAR
	{attribute addProperty Name "<#Heart beat#>"}
  	_heartBeat : BOOL;
	
	_iconSet: ARRAY[0..LAST_ICON_INDEX] OF Icon;

	_badgeValue : INT;
	
//~	
    _toggle: TcoUtilities.TcoBlinker(THIS^);
	
	_iconSetClear : ARRAY[0..LAST_ICON_INDEX] OF Icon; 
	
	_iconPlcPulse : Icon;
	
	_iconParamsClear : Icon;
	
	_currentIndex : INT;
//~
END_VAR



_iconPlcPulse.Title := '<#PLC connection#>';
_iconPlcPulse.IconType := TO_STRING(eIconType.plcConnection);
_iconPlcPulse.Signal := _heartBeat;
_iconPlcPulse.EnableRedIcon := FALSE;

_IconSet[_currentIndex] := _iconPlcPulse;

Blink();
CountSignals();

METHOD AddIcon : BOOL
VAR_INPUT
	inIcon : Icon;
END_VAR

VAR 
	_index : INT;
END_VAR
IF _currentIndex > LAST_ICON_INDEX THEN
	RETURN;
END_IF

_IconSet[_currentIndex] := inIcon;
_currentIndex := _currentIndex + 1;
END_METHOD

